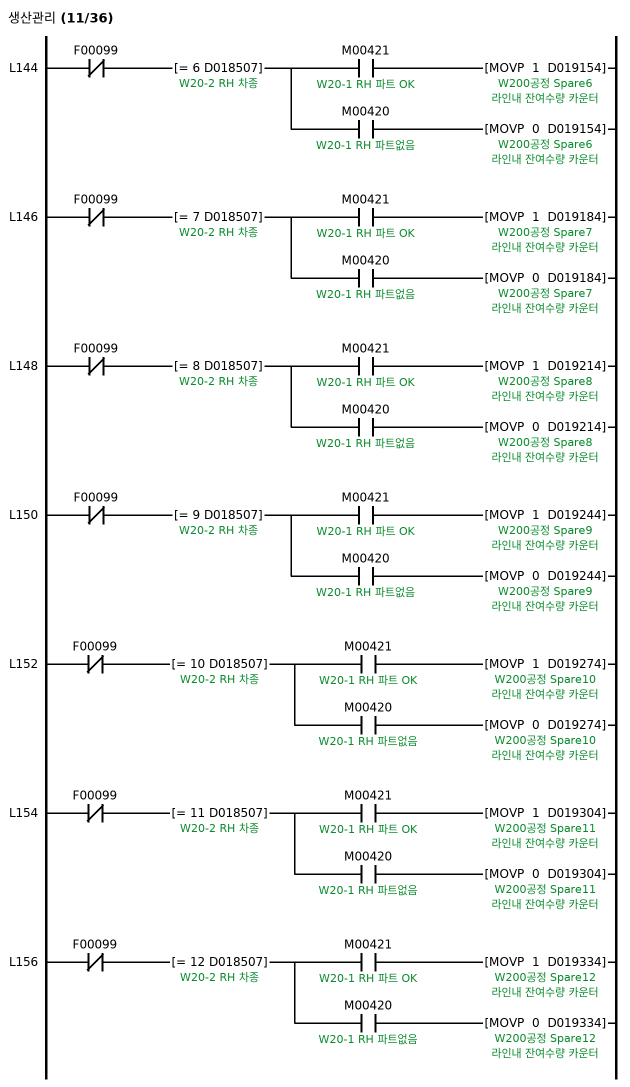
[picture p456: 생산관리 rungs L144-L156]
; L144
LOAD NOT  F00099
AND=      6 D018507	// W20-2 RH 차종
MPUSH
AND       M00421	// W20-1 RH 파트 OK
MOVP      1 D019154	// W200공정 Spare6 라인내 잔여수량 카운터
MPOP
AND       M00420	// W20-1 RH 파트없음
MOVP      0 D019154	// W200공정 Spare6 라인내 잔여수량 카운터
; L146
LOAD NOT  F00099
AND=      7 D018507	// W20-2 RH 차종
MPUSH
AND       M00421	// W20-1 RH 파트 OK
MOVP      1 D019184	// W200공정 Spare7 라인내 잔여수량 카운터
MPOP
AND       M00420	// W20-1 RH 파트없음
MOVP      0 D019184	// W200공정 Spare7 라인내 잔여수량 카운터
; L148
LOAD NOT  F00099
AND=      8 D018507	// W20-2 RH 차종
MPUSH
AND       M00421	// W20-1 RH 파트 OK
MOVP      1 D019214	// W200공정 Spare8 라인내 잔여수량 카운터
MPOP
AND       M00420	// W20-1 RH 파트없음
MOVP      0 D019214	// W200공정 Spare8 라인내 잔여수량 카운터
; L150
LOAD NOT  F00099
AND=      9 D018507	// W20-2 RH 차종
MPUSH
AND       M00421	// W20-1 RH 파트 OK
MOVP      1 D019244	// W200공정 Spare9 라인내 잔여수량 카운터
MPOP
AND       M00420	// W20-1 RH 파트없음
MOVP      0 D019244	// W200공정 Spare9 라인내 잔여수량 카운터
; L152
LOAD NOT  F00099
AND=      10 D018507	// W20-2 RH 차종
MPUSH
AND       M00421	// W20-1 RH 파트 OK
MOVP      1 D019274	// W200공정 Spare10 라인내 잔여수량 카운터
MPOP
AND       M00420	// W20-1 RH 파트없음
MOVP      0 D019274	// W200공정 Spare10 라인내 잔여수량 카운터
; L154
LOAD NOT  F00099
AND=      11 D018507	// W20-2 RH 차종
MPUSH
AND       M00421	// W20-1 RH 파트 OK
MOVP      1 D019304	// W200공정 Spare11 라인내 잔여수량 카운터
MPOP
AND       M00420	// W20-1 RH 파트없음
MOVP      0 D019304	// W200공정 Spare11 라인내 잔여수량 카운터
; L156
LOAD NOT  F00099
AND=      12 D018507	// W20-2 RH 차종
MPUSH
AND       M00421	// W20-1 RH 파트 OK
MOVP      1 D019334	// W200공정 Spare12 라인내 잔여수량 카운터
MPOP
AND       M00420	// W20-1 RH 파트없음
MOVP      0 D019334	// W200공정 Spare12 라인내 잔여수량 카운터

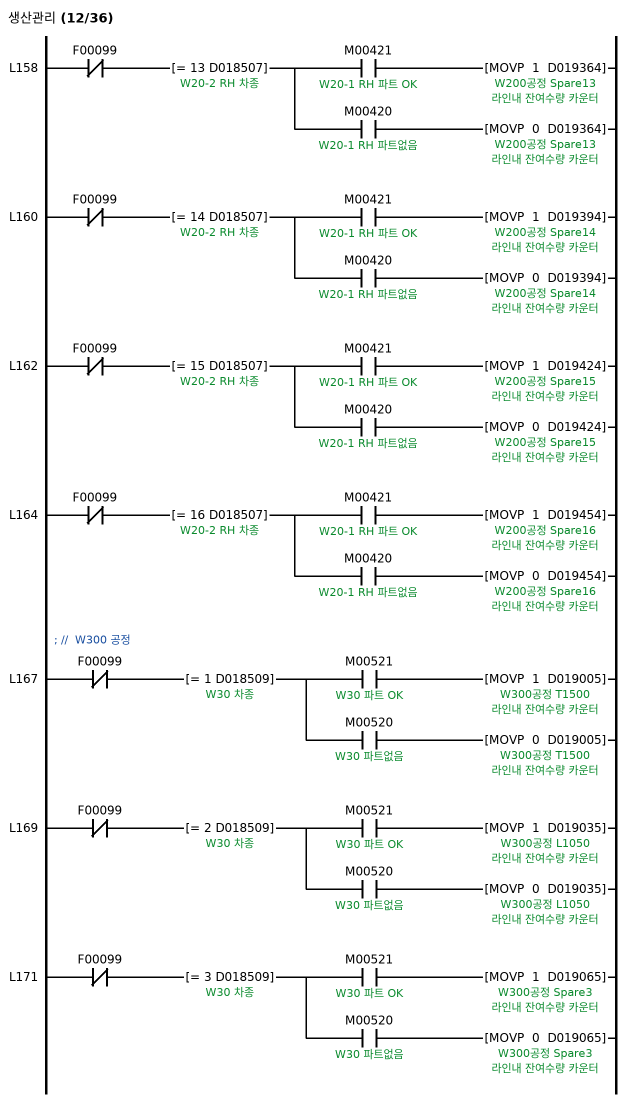
; L158
LOAD NOT  F00099
AND=      13 D018507	// W20-2 RH 차종
MPUSH
AND       M00421	// W20-1 RH 파트 OK
MOVP      1 D019364	// W200공정 Spare13 라인내 잔여수량 카운터
MPOP
AND       M00420	// W20-1 RH 파트없음
MOVP      0 D019364	// W200공정 Spare13 라인내 잔여수량 카운터
; L160
LOAD NOT  F00099
AND=      14 D018507	// W20-2 RH 차종
MPUSH
AND       M00421	// W20-1 RH 파트 OK
MOVP      1 D019394	// W200공정 Spare14 라인내 잔여수량 카운터
MPOP
AND       M00420	// W20-1 RH 파트없음
MOVP      0 D019394	// W200공정 Spare14 라인내 잔여수량 카운터
; L162
LOAD NOT  F00099
AND=      15 D018507	// W20-2 RH 차종
MPUSH
AND       M00421	// W20-1 RH 파트 OK
MOVP      1 D019424	// W200공정 Spare15 라인내 잔여수량 카운터
MPOP
AND       M00420	// W20-1 RH 파트없음
MOVP      0 D019424	// W200공정 Spare15 라인내 잔여수량 카운터
; L164
LOAD NOT  F00099
AND=      16 D018507	// W20-2 RH 차종
MPUSH
AND       M00421	// W20-1 RH 파트 OK
MOVP      1 D019454	// W200공정 Spare16 라인내 잔여수량 카운터
MPOP
AND       M00420	// W20-1 RH 파트없음
MOVP      0 D019454	// W200공정 Spare16 라인내 잔여수량 카운터
//   //  W300 공정
; L167
LOAD NOT  F00099
AND=      1 D018509	// W30 차종
MPUSH
AND       M00521	// W30 파트 OK
MOVP      1 D019005	// W300공정 T1500 라인내 잔여수량 카운터
MPOP
AND       M00520	// W30 파트없음
MOVP      0 D019005	// W300공정 T1500 라인내 잔여수량 카운터
; L169
LOAD NOT  F00099
AND=      2 D018509	// W30 차종
MPUSH
AND       M00521	// W30 파트 OK
MOVP      1 D019035	// W300공정 L1050 라인내 잔여수량 카운터
MPOP
AND       M00520	// W30 파트없음
MOVP      0 D019035	// W300공정 L1050 라인내 잔여수량 카운터
; L171
LOAD NOT  F00099
AND=      3 D018509	// W30 차종
MPUSH
AND       M00521	// W30 파트 OK
MOVP      1 D019065	// W300공정 Spare3 라인내 잔여수량 카운터
MPOP
AND       M00520	// W30 파트없음
MOVP      0 D019065	// W300공정 Spare3 라인내 잔여수량 카운터

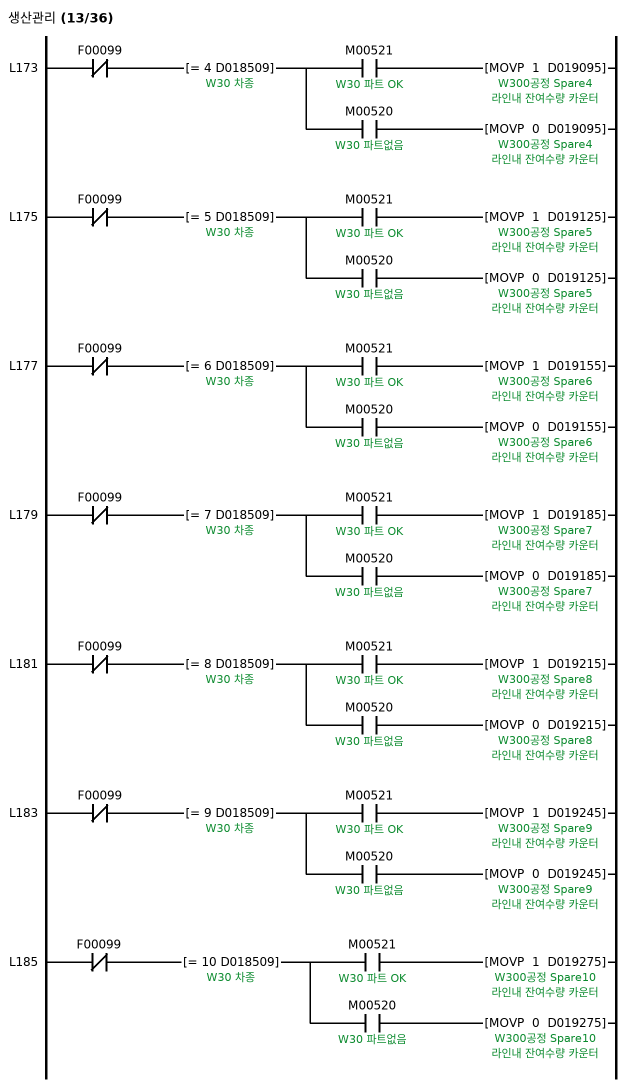
; L173
LOAD NOT  F00099
AND=      4 D018509	// W30 차종
MPUSH
AND       M00521	// W30 파트 OK
MOVP      1 D019095	// W300공정 Spare4 라인내 잔여수량 카운터
MPOP
AND       M00520	// W30 파트없음
MOVP      0 D019095	// W300공정 Spare4 라인내 잔여수량 카운터
; L175
LOAD NOT  F00099
AND=      5 D018509	// W30 차종
MPUSH
AND       M00521	// W30 파트 OK
MOVP      1 D019125	// W300공정 Spare5 라인내 잔여수량 카운터
MPOP
AND       M00520	// W30 파트없음
MOVP      0 D019125	// W300공정 Spare5 라인내 잔여수량 카운터
; L177
LOAD NOT  F00099
AND=      6 D018509	// W30 차종
MPUSH
AND       M00521	// W30 파트 OK
MOVP      1 D019155	// W300공정 Spare6 라인내 잔여수량 카운터
MPOP
AND       M00520	// W30 파트없음
MOVP      0 D019155	// W300공정 Spare6 라인내 잔여수량 카운터
; L179
LOAD NOT  F00099
AND=      7 D018509	// W30 차종
MPUSH
AND       M00521	// W30 파트 OK
MOVP      1 D019185	// W300공정 Spare7 라인내 잔여수량 카운터
MPOP
AND       M00520	// W30 파트없음
MOVP      0 D019185	// W300공정 Spare7 라인내 잔여수량 카운터
; L181
LOAD NOT  F00099
AND=      8 D018509	// W30 차종
MPUSH
AND       M00521	// W30 파트 OK
MOVP      1 D019215	// W300공정 Spare8 라인내 잔여수량 카운터
MPOP
AND       M00520	// W30 파트없음
MOVP      0 D019215	// W300공정 Spare8 라인내 잔여수량 카운터
; L183
LOAD NOT  F00099
AND=      9 D018509	// W30 차종
MPUSH
AND       M00521	// W30 파트 OK
MOVP      1 D019245	// W300공정 Spare9 라인내 잔여수량 카운터
MPOP
AND       M00520	// W30 파트없음
MOVP      0 D019245	// W300공정 Spare9 라인내 잔여수량 카운터
; L185
LOAD NOT  F00099
AND=      10 D018509	// W30 차종
MPUSH
AND       M00521	// W30 파트 OK
MOVP      1 D019275	// W300공정 Spare10 라인내 잔여수량 카운터
MPOP
AND       M00520	// W30 파트없음
MOVP      0 D019275	// W300공정 Spare10 라인내 잔여수량 카운터

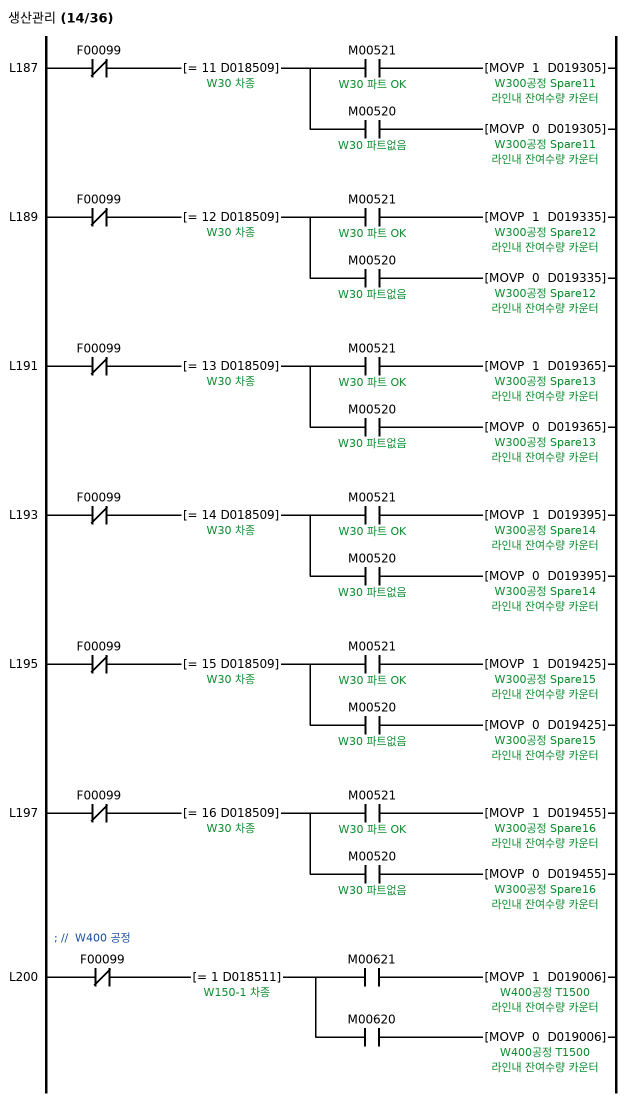
; L187
LOAD NOT  F00099
AND=      11 D018509	// W30 차종
MPUSH
AND       M00521	// W30 파트 OK
MOVP      1 D019305	// W300공정 Spare11 라인내 잔여수량 카운터
MPOP
AND       M00520	// W30 파트없음
MOVP      0 D019305	// W300공정 Spare11 라인내 잔여수량 카운터
; L189
LOAD NOT  F00099
AND=      12 D018509	// W30 차종
MPUSH
AND       M00521	// W30 파트 OK
MOVP      1 D019335	// W300공정 Spare12 라인내 잔여수량 카운터
MPOP
AND       M00520	// W30 파트없음
MOVP      0 D019335	// W300공정 Spare12 라인내 잔여수량 카운터
; L191
LOAD NOT  F00099
AND=      13 D018509	// W30 차종
MPUSH
AND       M00521	// W30 파트 OK
MOVP      1 D019365	// W300공정 Spare13 라인내 잔여수량 카운터
MPOP
AND       M00520	// W30 파트없음
MOVP      0 D019365	// W300공정 Spare13 라인내 잔여수량 카운터
; L193
LOAD NOT  F00099
AND=      14 D018509	// W30 차종
MPUSH
AND       M00521	// W30 파트 OK
MOVP      1 D019395	// W300공정 Spare14 라인내 잔여수량 카운터
MPOP
AND       M00520	// W30 파트없음
MOVP      0 D019395	// W300공정 Spare14 라인내 잔여수량 카운터
; L195
LOAD NOT  F00099
AND=      15 D018509	// W30 차종
MPUSH
AND       M00521	// W30 파트 OK
MOVP      1 D019425	// W300공정 Spare15 라인내 잔여수량 카운터
MPOP
AND       M00520	// W30 파트없음
MOVP      0 D019425	// W300공정 Spare15 라인내 잔여수량 카운터
; L197
LOAD NOT  F00099
AND=      16 D018509	// W30 차종
MPUSH
AND       M00521	// W30 파트 OK
MOVP      1 D019455	// W300공정 Spare16 라인내 잔여수량 카운터
MPOP
AND       M00520	// W30 파트없음
MOVP      0 D019455	// W300공정 Spare16 라인내 잔여수량 카운터
//   //  W400 공정
; L200
LOAD NOT  F00099
AND=      1 D018511	// W150-1 차종
MPUSH
AND       M00621
MOVP      1 D019006	// W400공정 T1500 라인내 잔여수량 카운터
MPOP
AND       M00620
MOVP      0 D019006	// W400공정 T1500 라인내 잔여수량 카운터

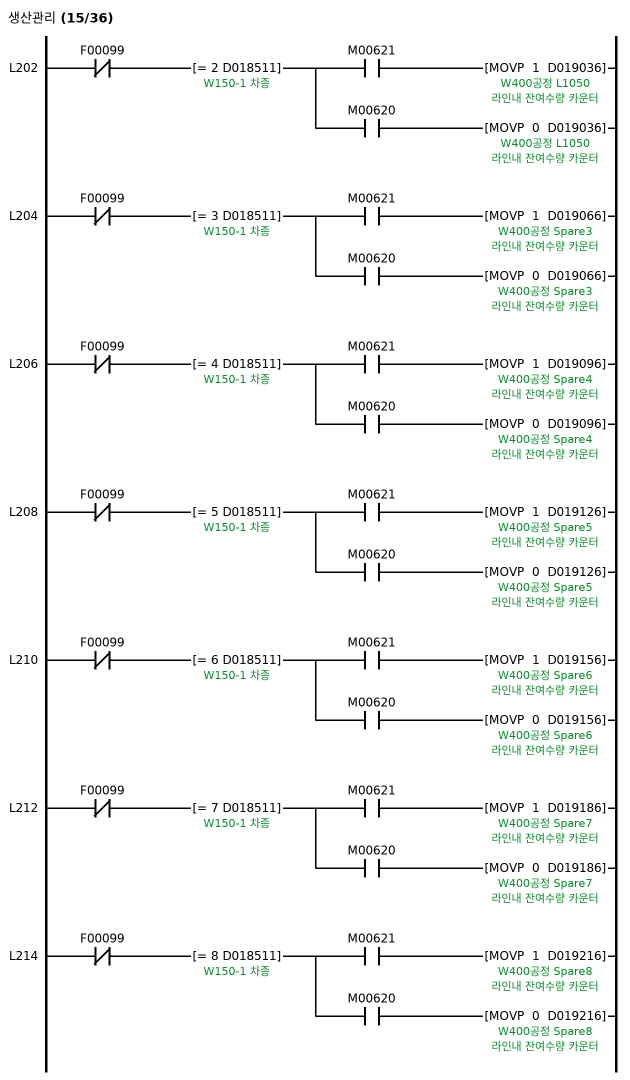
; L202
LOAD NOT  F00099
AND=      2 D018511	// W150-1 차종
MPUSH
AND       M00621
MOVP      1 D019036	// W400공정 L1050 라인내 잔여수량 카운터
MPOP
AND       M00620
MOVP      0 D019036	// W400공정 L1050 라인내 잔여수량 카운터
; L204
LOAD NOT  F00099
AND=      3 D018511	// W150-1 차종
MPUSH
AND       M00621
MOVP      1 D019066	// W400공정 Spare3 라인내 잔여수량 카운터
MPOP
AND       M00620
MOVP      0 D019066	// W400공정 Spare3 라인내 잔여수량 카운터
; L206
LOAD NOT  F00099
AND=      4 D018511	// W150-1 차종
MPUSH
AND       M00621
MOVP      1 D019096	// W400공정 Spare4 라인내 잔여수량 카운터
MPOP
AND       M00620
MOVP      0 D019096	// W400공정 Spare4 라인내 잔여수량 카운터
; L208
LOAD NOT  F00099
AND=      5 D018511	// W150-1 차종
MPUSH
AND       M00621
MOVP      1 D019126	// W400공정 Spare5 라인내 잔여수량 카운터
MPOP
AND       M00620
MOVP      0 D019126	// W400공정 Spare5 라인내 잔여수량 카운터
; L210
LOAD NOT  F00099
AND=      6 D018511	// W150-1 차종
MPUSH
AND       M00621
MOVP      1 D019156	// W400공정 Spare6 라인내 잔여수량 카운터
MPOP
AND       M00620
MOVP      0 D019156	// W400공정 Spare6 라인내 잔여수량 카운터
; L212
LOAD NOT  F00099
AND=      7 D018511	// W150-1 차종
MPUSH
AND       M00621
MOVP      1 D019186	// W400공정 Spare7 라인내 잔여수량 카운터
MPOP
AND       M00620
MOVP      0 D019186	// W400공정 Spare7 라인내 잔여수량 카운터
; L214
LOAD NOT  F00099
AND=      8 D018511	// W150-1 차종
MPUSH
AND       M00621
MOVP      1 D019216	// W400공정 Spare8 라인내 잔여수량 카운터
MPOP
AND       M00620
MOVP      0 D019216	// W400공정 Spare8 라인내 잔여수량 카운터

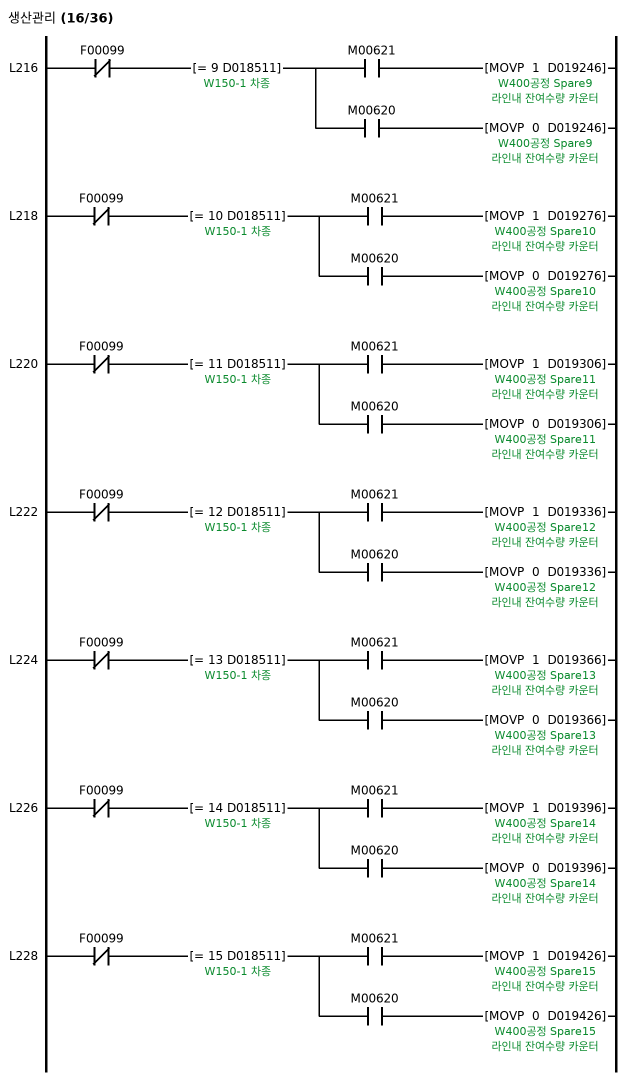
; L216
LOAD NOT  F00099
AND=      9 D018511	// W150-1 차종
MPUSH
AND       M00621
MOVP      1 D019246	// W400공정 Spare9 라인내 잔여수량 카운터
MPOP
AND       M00620
MOVP      0 D019246	// W400공정 Spare9 라인내 잔여수량 카운터
; L218
LOAD NOT  F00099
AND=      10 D018511	// W150-1 차종
MPUSH
AND       M00621
MOVP      1 D019276	// W400공정 Spare10 라인내 잔여수량 카운터
MPOP
AND       M00620
MOVP      0 D019276	// W400공정 Spare10 라인내 잔여수량 카운터
; L220
LOAD NOT  F00099
AND=      11 D018511	// W150-1 차종
MPUSH
AND       M00621
MOVP      1 D019306	// W400공정 Spare11 라인내 잔여수량 카운터
MPOP
AND       M00620
MOVP      0 D019306	// W400공정 Spare11 라인내 잔여수량 카운터
; L222
LOAD NOT  F00099
AND=      12 D018511	// W150-1 차종
MPUSH
AND       M00621
MOVP      1 D019336	// W400공정 Spare12 라인내 잔여수량 카운터
MPOP
AND       M00620
MOVP      0 D019336	// W400공정 Spare12 라인내 잔여수량 카운터
; L224
LOAD NOT  F00099
AND=      13 D018511	// W150-1 차종
MPUSH
AND       M00621
MOVP      1 D019366	// W400공정 Spare13 라인내 잔여수량 카운터
MPOP
AND       M00620
MOVP      0 D019366	// W400공정 Spare13 라인내 잔여수량 카운터
; L226
LOAD NOT  F00099
AND=      14 D018511	// W150-1 차종
MPUSH
AND       M00621
MOVP      1 D019396	// W400공정 Spare14 라인내 잔여수량 카운터
MPOP
AND       M00620
MOVP      0 D019396	// W400공정 Spare14 라인내 잔여수량 카운터
; L228
LOAD NOT  F00099
AND=      15 D018511	// W150-1 차종
MPUSH
AND       M00621
MOVP      1 D019426	// W400공정 Spare15 라인내 잔여수량 카운터
MPOP
AND       M00620
MOVP      0 D019426	// W400공정 Spare15 라인내 잔여수량 카운터

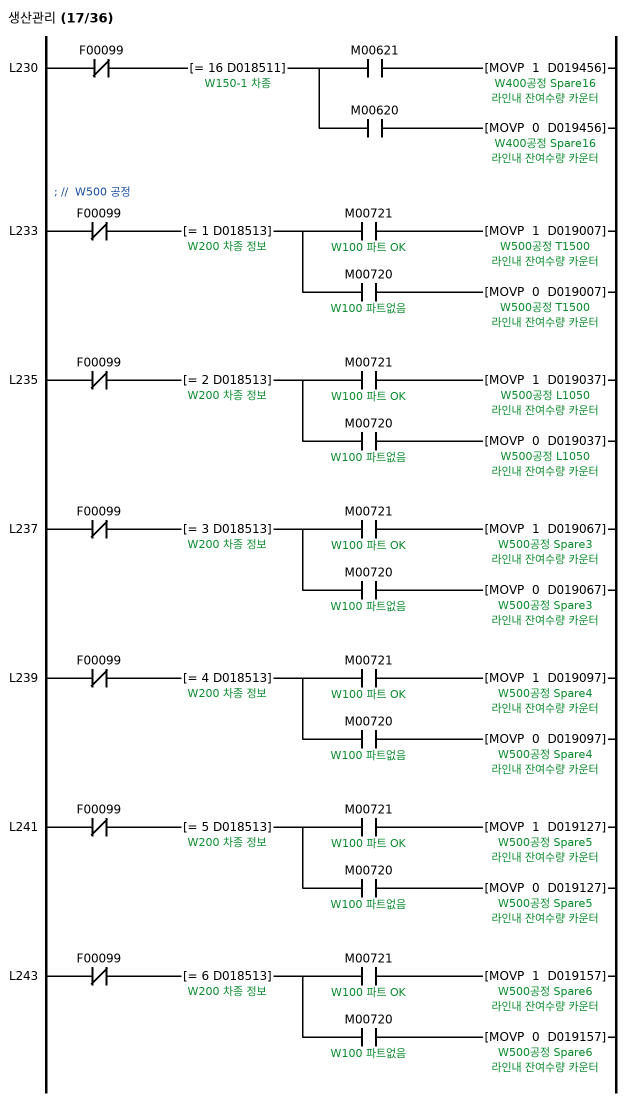
; L230
LOAD NOT  F00099
AND=      16 D018511	// W150-1 차종
MPUSH
AND       M00621
MOVP      1 D019456	// W400공정 Spare16 라인내 잔여수량 카운터
MPOP
AND       M00620
MOVP      0 D019456	// W400공정 Spare16 라인내 잔여수량 카운터
//   //  W500 공정
; L233
LOAD NOT  F00099
AND=      1 D018513	// W200 차종 정보
MPUSH
AND       M00721	// W100 파트 OK
MOVP      1 D019007	// W500공정 T1500 라인내 잔여수량 카운터
MPOP
AND       M00720	// W100 파트없음
MOVP      0 D019007	// W500공정 T1500 라인내 잔여수량 카운터
; L235
LOAD NOT  F00099
AND=      2 D018513	// W200 차종 정보
MPUSH
AND       M00721	// W100 파트 OK
MOVP      1 D019037	// W500공정 L1050 라인내 잔여수량 카운터
MPOP
AND       M00720	// W100 파트없음
MOVP      0 D019037	// W500공정 L1050 라인내 잔여수량 카운터
; L237
LOAD NOT  F00099
AND=      3 D018513	// W200 차종 정보
MPUSH
AND       M00721	// W100 파트 OK
MOVP      1 D019067	// W500공정 Spare3 라인내 잔여수량 카운터
MPOP
AND       M00720	// W100 파트없음
MOVP      0 D019067	// W500공정 Spare3 라인내 잔여수량 카운터
; L239
LOAD NOT  F00099
AND=      4 D018513	// W200 차종 정보
MPUSH
AND       M00721	// W100 파트 OK
MOVP      1 D019097	// W500공정 Spare4 라인내 잔여수량 카운터
MPOP
AND       M00720	// W100 파트없음
MOVP      0 D019097	// W500공정 Spare4 라인내 잔여수량 카운터
; L241
LOAD NOT  F00099
AND=      5 D018513	// W200 차종 정보
MPUSH
AND       M00721	// W100 파트 OK
MOVP      1 D019127	// W500공정 Spare5 라인내 잔여수량 카운터
MPOP
AND       M00720	// W100 파트없음
MOVP      0 D019127	// W500공정 Spare5 라인내 잔여수량 카운터
; L243
LOAD NOT  F00099
AND=      6 D018513	// W200 차종 정보
MPUSH
AND       M00721	// W100 파트 OK
MOVP      1 D019157	// W500공정 Spare6 라인내 잔여수량 카운터
MPOP
AND       M00720	// W100 파트없음
MOVP      0 D019157	// W500공정 Spare6 라인내 잔여수량 카운터

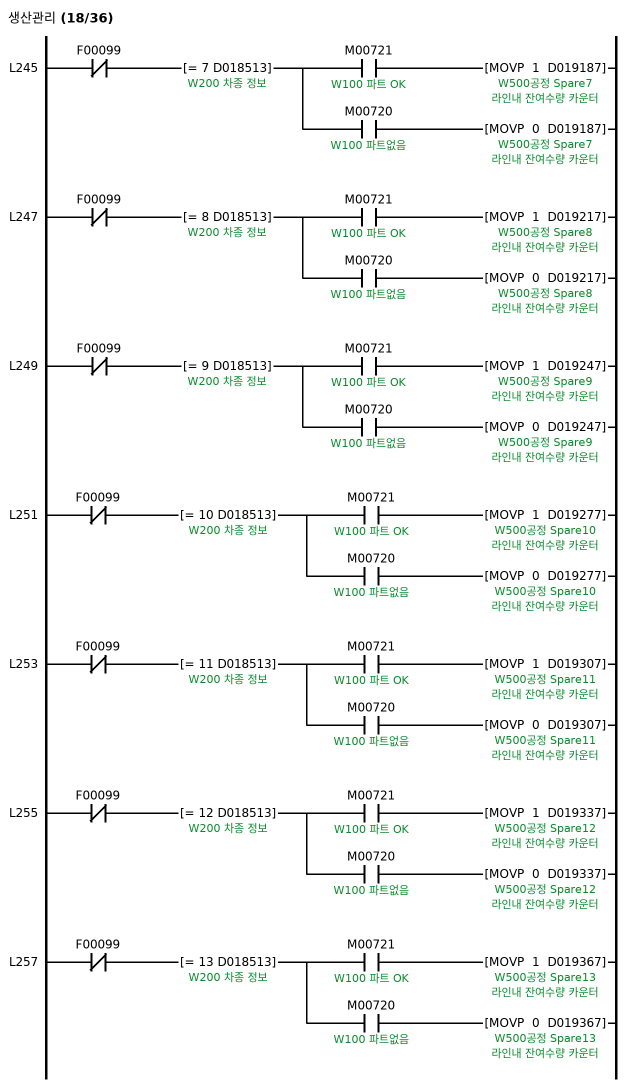
; L245
LOAD NOT  F00099
AND=      7 D018513	// W200 차종 정보
MPUSH
AND       M00721	// W100 파트 OK
MOVP      1 D019187	// W500공정 Spare7 라인내 잔여수량 카운터
MPOP
AND       M00720	// W100 파트없음
MOVP      0 D019187	// W500공정 Spare7 라인내 잔여수량 카운터
; L247
LOAD NOT  F00099
AND=      8 D018513	// W200 차종 정보
MPUSH
AND       M00721	// W100 파트 OK
MOVP      1 D019217	// W500공정 Spare8 라인내 잔여수량 카운터
MPOP
AND       M00720	// W100 파트없음
MOVP      0 D019217	// W500공정 Spare8 라인내 잔여수량 카운터
; L249
LOAD NOT  F00099
AND=      9 D018513	// W200 차종 정보
MPUSH
AND       M00721	// W100 파트 OK
MOVP      1 D019247	// W500공정 Spare9 라인내 잔여수량 카운터
MPOP
AND       M00720	// W100 파트없음
MOVP      0 D019247	// W500공정 Spare9 라인내 잔여수량 카운터
; L251
LOAD NOT  F00099
AND=      10 D018513	// W200 차종 정보
MPUSH
AND       M00721	// W100 파트 OK
MOVP      1 D019277	// W500공정 Spare10 라인내 잔여수량 카운터
MPOP
AND       M00720	// W100 파트없음
MOVP      0 D019277	// W500공정 Spare10 라인내 잔여수량 카운터
; L253
LOAD NOT  F00099
AND=      11 D018513	// W200 차종 정보
MPUSH
AND       M00721	// W100 파트 OK
MOVP      1 D019307	// W500공정 Spare11 라인내 잔여수량 카운터
MPOP
AND       M00720	// W100 파트없음
MOVP      0 D019307	// W500공정 Spare11 라인내 잔여수량 카운터
; L255
LOAD NOT  F00099
AND=      12 D018513	// W200 차종 정보
MPUSH
AND       M00721	// W100 파트 OK
MOVP      1 D019337	// W500공정 Spare12 라인내 잔여수량 카운터
MPOP
AND       M00720	// W100 파트없음
MOVP      0 D019337	// W500공정 Spare12 라인내 잔여수량 카운터
; L257
LOAD NOT  F00099
AND=      13 D018513	// W200 차종 정보
MPUSH
AND       M00721	// W100 파트 OK
MOVP      1 D019367	// W500공정 Spare13 라인내 잔여수량 카운터
MPOP
AND       M00720	// W100 파트없음
MOVP      0 D019367	// W500공정 Spare13 라인내 잔여수량 카운터

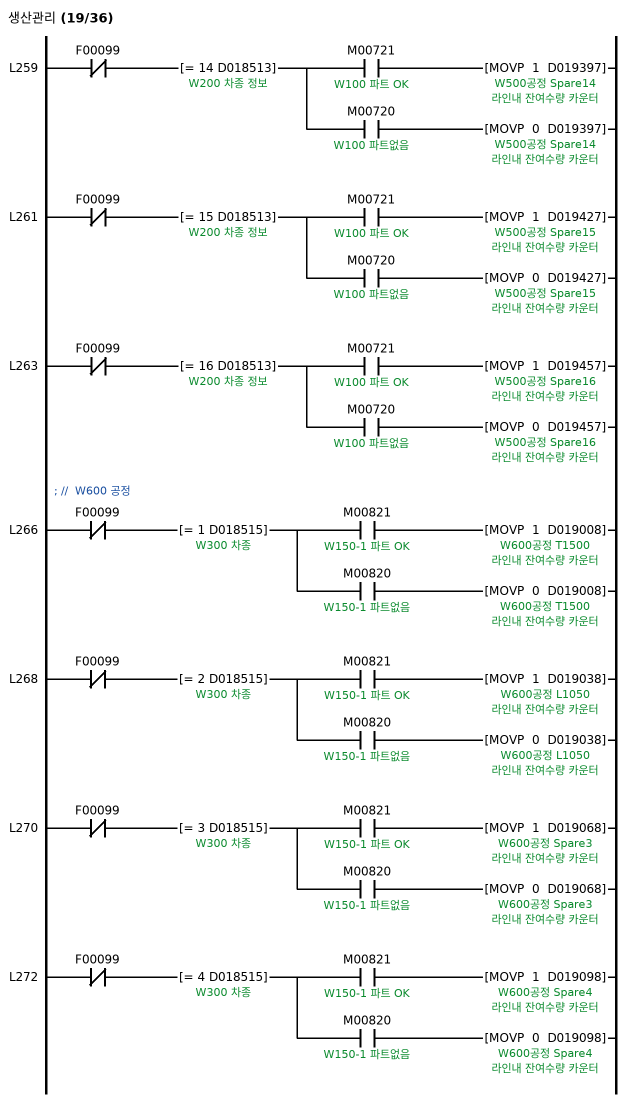
; L259
LOAD NOT  F00099
AND=      14 D018513	// W200 차종 정보
MPUSH
AND       M00721	// W100 파트 OK
MOVP      1 D019397	// W500공정 Spare14 라인내 잔여수량 카운터
MPOP
AND       M00720	// W100 파트없음
MOVP      0 D019397	// W500공정 Spare14 라인내 잔여수량 카운터
; L261
LOAD NOT  F00099
AND=      15 D018513	// W200 차종 정보
MPUSH
AND       M00721	// W100 파트 OK
MOVP      1 D019427	// W500공정 Spare15 라인내 잔여수량 카운터
MPOP
AND       M00720	// W100 파트없음
MOVP      0 D019427	// W500공정 Spare15 라인내 잔여수량 카운터
; L263
LOAD NOT  F00099
AND=      16 D018513	// W200 차종 정보
MPUSH
AND       M00721	// W100 파트 OK
MOVP      1 D019457	// W500공정 Spare16 라인내 잔여수량 카운터
MPOP
AND       M00720	// W100 파트없음
MOVP      0 D019457	// W500공정 Spare16 라인내 잔여수량 카운터
//   //  W600 공정
; L266
LOAD NOT  F00099
AND=      1 D018515	// W300 차종
MPUSH
AND       M00821	// W150-1 파트 OK
MOVP      1 D019008	// W600공정 T1500 라인내 잔여수량 카운터
MPOP
AND       M00820	// W150-1 파트없음
MOVP      0 D019008	// W600공정 T1500 라인내 잔여수량 카운터
; L268
LOAD NOT  F00099
AND=      2 D018515	// W300 차종
MPUSH
AND       M00821	// W150-1 파트 OK
MOVP      1 D019038	// W600공정 L1050 라인내 잔여수량 카운터
MPOP
AND       M00820	// W150-1 파트없음
MOVP      0 D019038	// W600공정 L1050 라인내 잔여수량 카운터
; L270
LOAD NOT  F00099
AND=      3 D018515	// W300 차종
MPUSH
AND       M00821	// W150-1 파트 OK
MOVP      1 D019068	// W600공정 Spare3 라인내 잔여수량 카운터
MPOP
AND       M00820	// W150-1 파트없음
MOVP      0 D019068	// W600공정 Spare3 라인내 잔여수량 카운터
; L272
LOAD NOT  F00099
AND=      4 D018515	// W300 차종
MPUSH
AND       M00821	// W150-1 파트 OK
MOVP      1 D019098	// W600공정 Spare4 라인내 잔여수량 카운터
MPOP
AND       M00820	// W150-1 파트없음
MOVP      0 D019098	// W600공정 Spare4 라인내 잔여수량 카운터

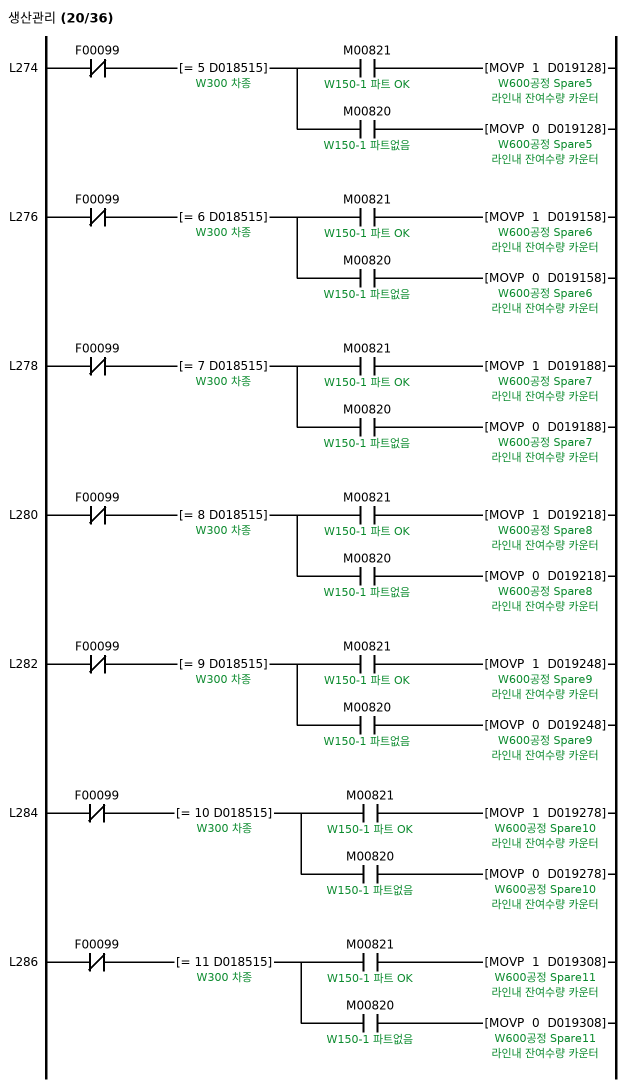
; L274
LOAD NOT  F00099
AND=      5 D018515	// W300 차종
MPUSH
AND       M00821	// W150-1 파트 OK
MOVP      1 D019128	// W600공정 Spare5 라인내 잔여수량 카운터
MPOP
AND       M00820	// W150-1 파트없음
MOVP      0 D019128	// W600공정 Spare5 라인내 잔여수량 카운터
; L276
LOAD NOT  F00099
AND=      6 D018515	// W300 차종
MPUSH
AND       M00821	// W150-1 파트 OK
MOVP      1 D019158	// W600공정 Spare6 라인내 잔여수량 카운터
MPOP
AND       M00820	// W150-1 파트없음
MOVP      0 D019158	// W600공정 Spare6 라인내 잔여수량 카운터
; L278
LOAD NOT  F00099
AND=      7 D018515	// W300 차종
MPUSH
AND       M00821	// W150-1 파트 OK
MOVP      1 D019188	// W600공정 Spare7 라인내 잔여수량 카운터
MPOP
AND       M00820	// W150-1 파트없음
MOVP      0 D019188	// W600공정 Spare7 라인내 잔여수량 카운터
; L280
LOAD NOT  F00099
AND=      8 D018515	// W300 차종
MPUSH
AND       M00821	// W150-1 파트 OK
MOVP      1 D019218	// W600공정 Spare8 라인내 잔여수량 카운터
MPOP
AND       M00820	// W150-1 파트없음
MOVP      0 D019218	// W600공정 Spare8 라인내 잔여수량 카운터
; L282
LOAD NOT  F00099
AND=      9 D018515	// W300 차종
MPUSH
AND       M00821	// W150-1 파트 OK
MOVP      1 D019248	// W600공정 Spare9 라인내 잔여수량 카운터
MPOP
AND       M00820	// W150-1 파트없음
MOVP      0 D019248	// W600공정 Spare9 라인내 잔여수량 카운터
; L284
LOAD NOT  F00099
AND=      10 D018515	// W300 차종
MPUSH
AND       M00821	// W150-1 파트 OK
MOVP      1 D019278	// W600공정 Spare10 라인내 잔여수량 카운터
MPOP
AND       M00820	// W150-1 파트없음
MOVP      0 D019278	// W600공정 Spare10 라인내 잔여수량 카운터
; L286
LOAD NOT  F00099
AND=      11 D018515	// W300 차종
MPUSH
AND       M00821	// W150-1 파트 OK
MOVP      1 D019308	// W600공정 Spare11 라인내 잔여수량 카운터
MPOP
AND       M00820	// W150-1 파트없음
MOVP      0 D019308	// W600공정 Spare11 라인내 잔여수량 카운터

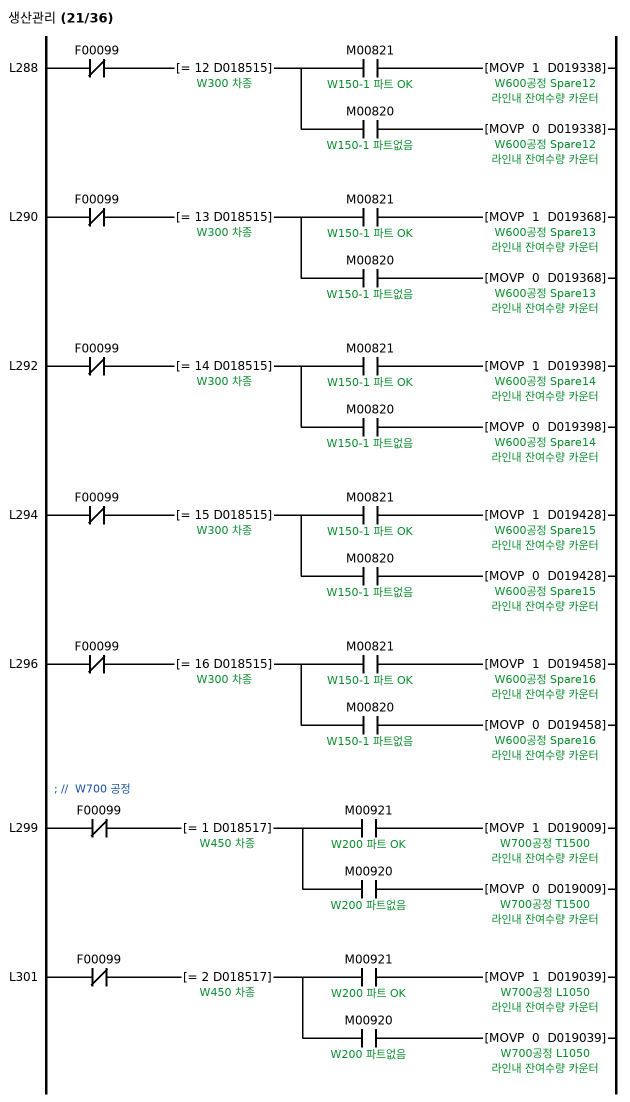
; L288
LOAD NOT  F00099
AND=      12 D018515	// W300 차종
MPUSH
AND       M00821	// W150-1 파트 OK
MOVP      1 D019338	// W600공정 Spare12 라인내 잔여수량 카운터
MPOP
AND       M00820	// W150-1 파트없음
MOVP      0 D019338	// W600공정 Spare12 라인내 잔여수량 카운터
; L290
LOAD NOT  F00099
AND=      13 D018515	// W300 차종
MPUSH
AND       M00821	// W150-1 파트 OK
MOVP      1 D019368	// W600공정 Spare13 라인내 잔여수량 카운터
MPOP
AND       M00820	// W150-1 파트없음
MOVP      0 D019368	// W600공정 Spare13 라인내 잔여수량 카운터
; L292
LOAD NOT  F00099
AND=      14 D018515	// W300 차종
MPUSH
AND       M00821	// W150-1 파트 OK
MOVP      1 D019398	// W600공정 Spare14 라인내 잔여수량 카운터
MPOP
AND       M00820	// W150-1 파트없음
MOVP      0 D019398	// W600공정 Spare14 라인내 잔여수량 카운터
; L294
LOAD NOT  F00099
AND=      15 D018515	// W300 차종
MPUSH
AND       M00821	// W150-1 파트 OK
MOVP      1 D019428	// W600공정 Spare15 라인내 잔여수량 카운터
MPOP
AND       M00820	// W150-1 파트없음
MOVP      0 D019428	// W600공정 Spare15 라인내 잔여수량 카운터
; L296
LOAD NOT  F00099
AND=      16 D018515	// W300 차종
MPUSH
AND       M00821	// W150-1 파트 OK
MOVP      1 D019458	// W600공정 Spare16 라인내 잔여수량 카운터
MPOP
AND       M00820	// W150-1 파트없음
MOVP      0 D019458	// W600공정 Spare16 라인내 잔여수량 카운터
//   //  W700 공정
; L299
LOAD NOT  F00099
AND=      1 D018517	// W450 차종
MPUSH
AND       M00921	// W200 파트 OK
MOVP      1 D019009	// W700공정 T1500 라인내 잔여수량 카운터
MPOP
AND       M00920	// W200 파트없음
MOVP      0 D019009	// W700공정 T1500 라인내 잔여수량 카운터
; L301
LOAD NOT  F00099
AND=      2 D018517	// W450 차종
MPUSH
AND       M00921	// W200 파트 OK
MOVP      1 D019039	// W700공정 L1050 라인내 잔여수량 카운터
MPOP
AND       M00920	// W200 파트없음
MOVP      0 D019039	// W700공정 L1050 라인내 잔여수량 카운터

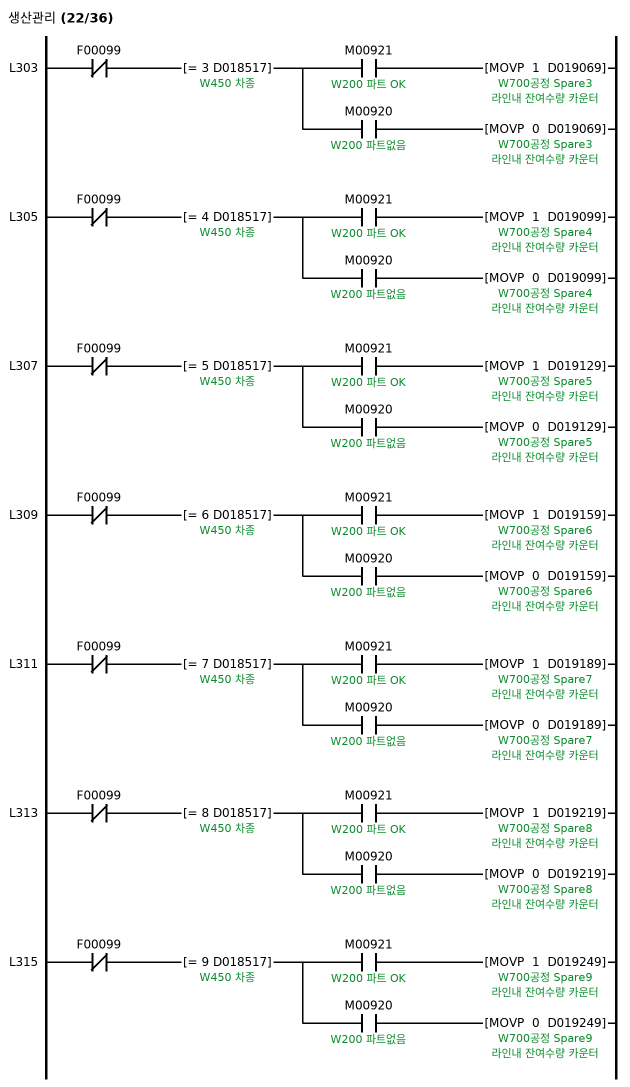
; L303
LOAD NOT  F00099
AND=      3 D018517	// W450 차종
MPUSH
AND       M00921	// W200 파트 OK
MOVP      1 D019069	// W700공정 Spare3 라인내 잔여수량 카운터
MPOP
AND       M00920	// W200 파트없음
MOVP      0 D019069	// W700공정 Spare3 라인내 잔여수량 카운터
; L305
LOAD NOT  F00099
AND=      4 D018517	// W450 차종
MPUSH
AND       M00921	// W200 파트 OK
MOVP      1 D019099	// W700공정 Spare4 라인내 잔여수량 카운터
MPOP
AND       M00920	// W200 파트없음
MOVP      0 D019099	// W700공정 Spare4 라인내 잔여수량 카운터
; L307
LOAD NOT  F00099
AND=      5 D018517	// W450 차종
MPUSH
AND       M00921	// W200 파트 OK
MOVP      1 D019129	// W700공정 Spare5 라인내 잔여수량 카운터
MPOP
AND       M00920	// W200 파트없음
MOVP      0 D019129	// W700공정 Spare5 라인내 잔여수량 카운터
; L309
LOAD NOT  F00099
AND=      6 D018517	// W450 차종
MPUSH
AND       M00921	// W200 파트 OK
MOVP      1 D019159	// W700공정 Spare6 라인내 잔여수량 카운터
MPOP
AND       M00920	// W200 파트없음
MOVP      0 D019159	// W700공정 Spare6 라인내 잔여수량 카운터
; L311
LOAD NOT  F00099
AND=      7 D018517	// W450 차종
MPUSH
AND       M00921	// W200 파트 OK
MOVP      1 D019189	// W700공정 Spare7 라인내 잔여수량 카운터
MPOP
AND       M00920	// W200 파트없음
MOVP      0 D019189	// W700공정 Spare7 라인내 잔여수량 카운터
; L313
LOAD NOT  F00099
AND=      8 D018517	// W450 차종
MPUSH
AND       M00921	// W200 파트 OK
MOVP      1 D019219	// W700공정 Spare8 라인내 잔여수량 카운터
MPOP
AND       M00920	// W200 파트없음
MOVP      0 D019219	// W700공정 Spare8 라인내 잔여수량 카운터
; L315
LOAD NOT  F00099
AND=      9 D018517	// W450 차종
MPUSH
AND       M00921	// W200 파트 OK
MOVP      1 D019249	// W700공정 Spare9 라인내 잔여수량 카운터
MPOP
AND       M00920	// W200 파트없음
MOVP      0 D019249	// W700공정 Spare9 라인내 잔여수량 카운터

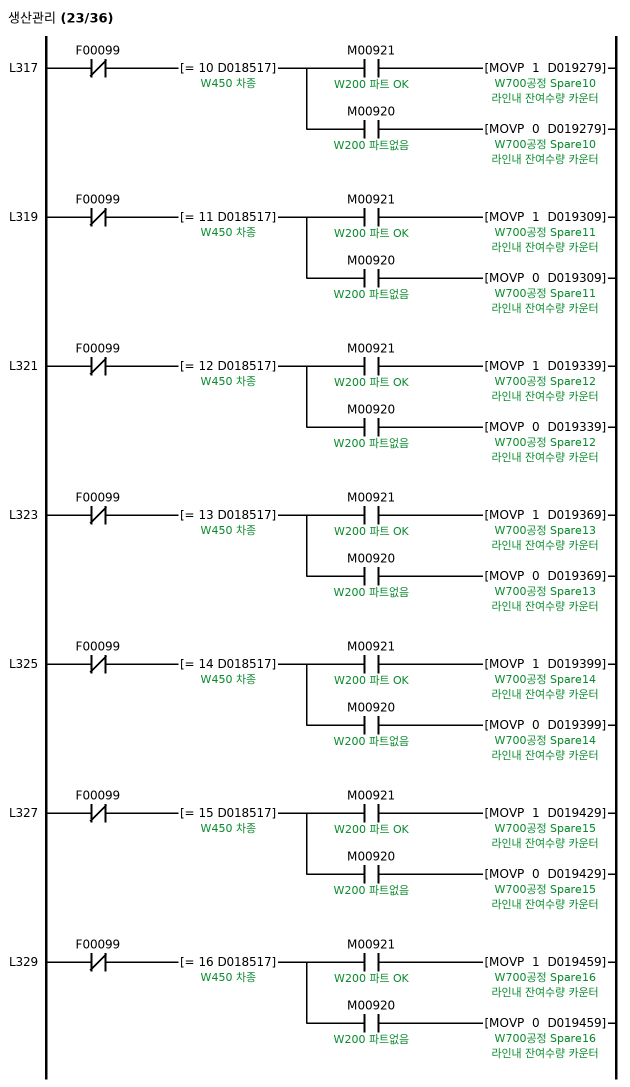
; L317
LOAD NOT  F00099
AND=      10 D018517	// W450 차종
MPUSH
AND       M00921	// W200 파트 OK
MOVP      1 D019279	// W700공정 Spare10 라인내 잔여수량 카운터
MPOP
AND       M00920	// W200 파트없음
MOVP      0 D019279	// W700공정 Spare10 라인내 잔여수량 카운터
; L319
LOAD NOT  F00099
AND=      11 D018517	// W450 차종
MPUSH
AND       M00921	// W200 파트 OK
MOVP      1 D019309	// W700공정 Spare11 라인내 잔여수량 카운터
MPOP
AND       M00920	// W200 파트없음
MOVP      0 D019309	// W700공정 Spare11 라인내 잔여수량 카운터
; L321
LOAD NOT  F00099
AND=      12 D018517	// W450 차종
MPUSH
AND       M00921	// W200 파트 OK
MOVP      1 D019339	// W700공정 Spare12 라인내 잔여수량 카운터
MPOP
AND       M00920	// W200 파트없음
MOVP      0 D019339	// W700공정 Spare12 라인내 잔여수량 카운터
; L323
LOAD NOT  F00099
AND=      13 D018517	// W450 차종
MPUSH
AND       M00921	// W200 파트 OK
MOVP      1 D019369	// W700공정 Spare13 라인내 잔여수량 카운터
MPOP
AND       M00920	// W200 파트없음
MOVP      0 D019369	// W700공정 Spare13 라인내 잔여수량 카운터
; L325
LOAD NOT  F00099
AND=      14 D018517	// W450 차종
MPUSH
AND       M00921	// W200 파트 OK
MOVP      1 D019399	// W700공정 Spare14 라인내 잔여수량 카운터
MPOP
AND       M00920	// W200 파트없음
MOVP      0 D019399	// W700공정 Spare14 라인내 잔여수량 카운터
; L327
LOAD NOT  F00099
AND=      15 D018517	// W450 차종
MPUSH
AND       M00921	// W200 파트 OK
MOVP      1 D019429	// W700공정 Spare15 라인내 잔여수량 카운터
MPOP
AND       M00920	// W200 파트없음
MOVP      0 D019429	// W700공정 Spare15 라인내 잔여수량 카운터
; L329
LOAD NOT  F00099
AND=      16 D018517	// W450 차종
MPUSH
AND       M00921	// W200 파트 OK
MOVP      1 D019459	// W700공정 Spare16 라인내 잔여수량 카운터
MPOP
AND       M00920	// W200 파트없음
MOVP      0 D019459	// W700공정 Spare16 라인내 잔여수량 카운터

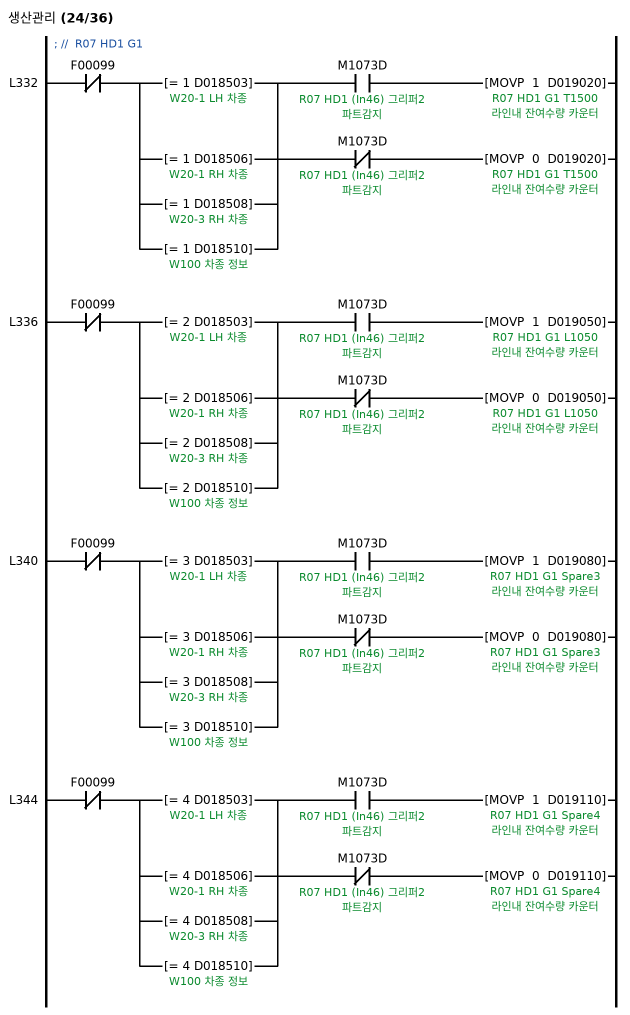
//   //  R07 HD1 G1
; L332
LOAD NOT  F00099
LOAD=     1 D018503	// W20-1 LH 차종
OR=       1 D018506	// W20-1 RH 차종
OR=       1 D018508	// W20-3 RH 차종
OR=       1 D018510	// W100 차종 정보
AND LOAD
MPUSH
AND       M1073D	// R07 HD1 (In46) 그리퍼2 파트감지
MOVP      1 D019020	// R07 HD1 G1 T1500 라인내 잔여수량 카운터
MPOP
AND NOT   M1073D	// R07 HD1 (In46) 그리퍼2 파트감지
MOVP      0 D019020	// R07 HD1 G1 T1500 라인내 잔여수량 카운터
; L336
LOAD NOT  F00099
LOAD=     2 D018503	// W20-1 LH 차종
OR=       2 D018506	// W20-1 RH 차종
OR=       2 D018508	// W20-3 RH 차종
OR=       2 D018510	// W100 차종 정보
AND LOAD
MPUSH
AND       M1073D	// R07 HD1 (In46) 그리퍼2 파트감지
MOVP      1 D019050	// R07 HD1 G1 L1050 라인내 잔여수량 카운터
MPOP
AND NOT   M1073D	// R07 HD1 (In46) 그리퍼2 파트감지
MOVP      0 D019050	// R07 HD1 G1 L1050 라인내 잔여수량 카운터
; L340
LOAD NOT  F00099
LOAD=     3 D018503	// W20-1 LH 차종
OR=       3 D018506	// W20-1 RH 차종
OR=       3 D018508	// W20-3 RH 차종
OR=       3 D018510	// W100 차종 정보
AND LOAD
MPUSH
AND       M1073D	// R07 HD1 (In46) 그리퍼2 파트감지
MOVP      1 D019080	// R07 HD1 G1 Spare3 라인내 잔여수량 카운터
MPOP
AND NOT   M1073D	// R07 HD1 (In46) 그리퍼2 파트감지
MOVP      0 D019080	// R07 HD1 G1 Spare3 라인내 잔여수량 카운터
; L344
LOAD NOT  F00099
LOAD=     4 D018503	// W20-1 LH 차종
OR=       4 D018506	// W20-1 RH 차종
OR=       4 D018508	// W20-3 RH 차종
OR=       4 D018510	// W100 차종 정보
AND LOAD
MPUSH
AND       M1073D	// R07 HD1 (In46) 그리퍼2 파트감지
MOVP      1 D019110	// R07 HD1 G1 Spare4 라인내 잔여수량 카운터
MPOP
AND NOT   M1073D	// R07 HD1 (In46) 그리퍼2 파트감지
MOVP      0 D019110	// R07 HD1 G1 Spare4 라인내 잔여수량 카운터

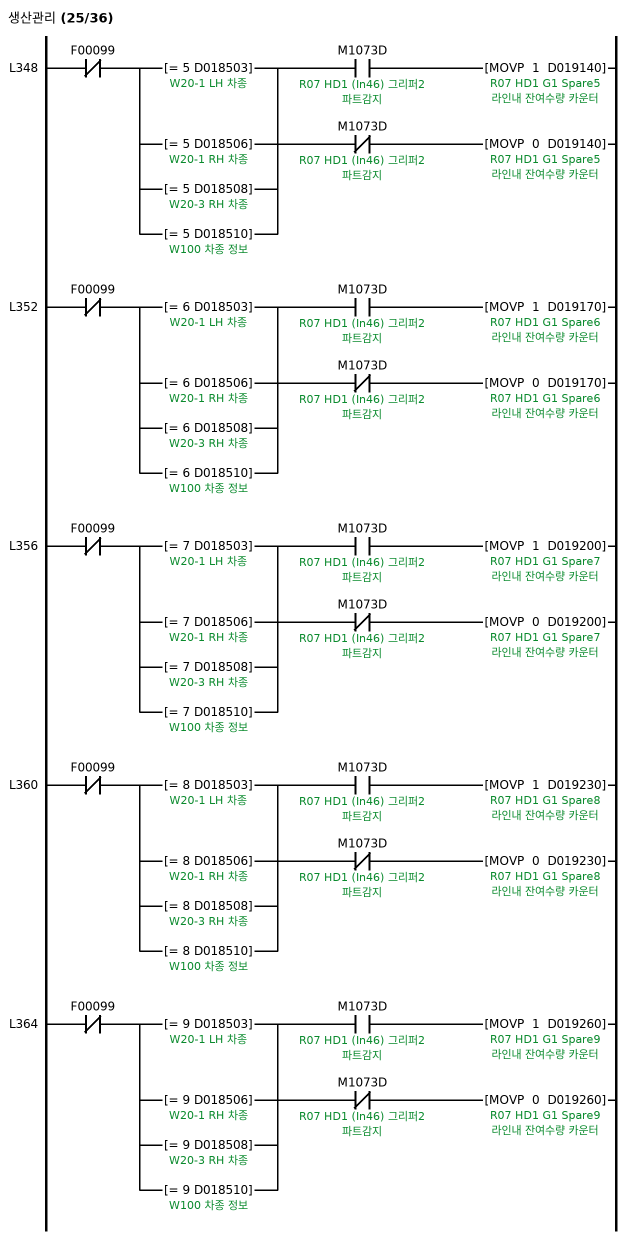
; L348
LOAD NOT  F00099
LOAD=     5 D018503	// W20-1 LH 차종
OR=       5 D018506	// W20-1 RH 차종
OR=       5 D018508	// W20-3 RH 차종
OR=       5 D018510	// W100 차종 정보
AND LOAD
MPUSH
AND       M1073D	// R07 HD1 (In46) 그리퍼2 파트감지
MOVP      1 D019140	// R07 HD1 G1 Spare5 라인내 잔여수량 카운터
MPOP
AND NOT   M1073D	// R07 HD1 (In46) 그리퍼2 파트감지
MOVP      0 D019140	// R07 HD1 G1 Spare5 라인내 잔여수량 카운터
; L352
LOAD NOT  F00099
LOAD=     6 D018503	// W20-1 LH 차종
OR=       6 D018506	// W20-1 RH 차종
OR=       6 D018508	// W20-3 RH 차종
OR=       6 D018510	// W100 차종 정보
AND LOAD
MPUSH
AND       M1073D	// R07 HD1 (In46) 그리퍼2 파트감지
MOVP      1 D019170	// R07 HD1 G1 Spare6 라인내 잔여수량 카운터
MPOP
AND NOT   M1073D	// R07 HD1 (In46) 그리퍼2 파트감지
MOVP      0 D019170	// R07 HD1 G1 Spare6 라인내 잔여수량 카운터
; L356
LOAD NOT  F00099
LOAD=     7 D018503	// W20-1 LH 차종
OR=       7 D018506	// W20-1 RH 차종
OR=       7 D018508	// W20-3 RH 차종
OR=       7 D018510	// W100 차종 정보
AND LOAD
MPUSH
AND       M1073D	// R07 HD1 (In46) 그리퍼2 파트감지
MOVP      1 D019200	// R07 HD1 G1 Spare7 라인내 잔여수량 카운터
MPOP
AND NOT   M1073D	// R07 HD1 (In46) 그리퍼2 파트감지
MOVP      0 D019200	// R07 HD1 G1 Spare7 라인내 잔여수량 카운터
; L360
LOAD NOT  F00099
LOAD=     8 D018503	// W20-1 LH 차종
OR=       8 D018506	// W20-1 RH 차종
OR=       8 D018508	// W20-3 RH 차종
OR=       8 D018510	// W100 차종 정보
AND LOAD
MPUSH
AND       M1073D	// R07 HD1 (In46) 그리퍼2 파트감지
MOVP      1 D019230	// R07 HD1 G1 Spare8 라인내 잔여수량 카운터
MPOP
AND NOT   M1073D	// R07 HD1 (In46) 그리퍼2 파트감지
MOVP      0 D019230	// R07 HD1 G1 Spare8 라인내 잔여수량 카운터
; L364
LOAD NOT  F00099
LOAD=     9 D018503	// W20-1 LH 차종
OR=       9 D018506	// W20-1 RH 차종
OR=       9 D018508	// W20-3 RH 차종
OR=       9 D018510	// W100 차종 정보
AND LOAD
MPUSH
AND       M1073D	// R07 HD1 (In46) 그리퍼2 파트감지
MOVP      1 D019260	// R07 HD1 G1 Spare9 라인내 잔여수량 카운터
MPOP
AND NOT   M1073D	// R07 HD1 (In46) 그리퍼2 파트감지
MOVP      0 D019260	// R07 HD1 G1 Spare9 라인내 잔여수량 카운터

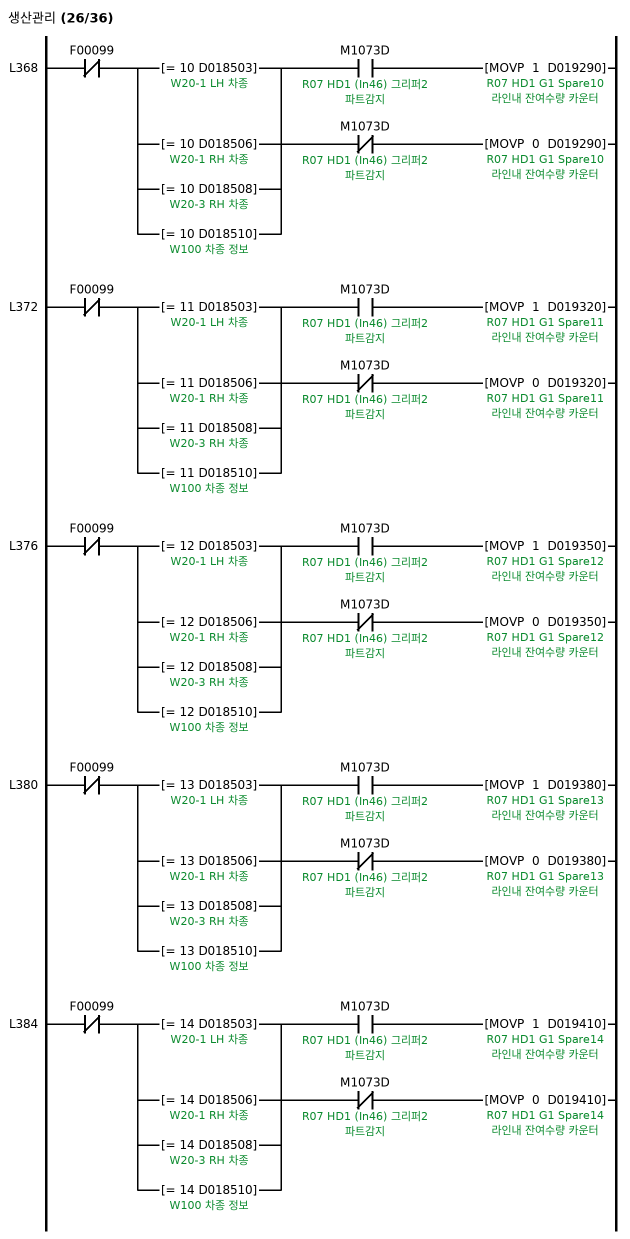
; L368
LOAD NOT  F00099
LOAD=     10 D018503	// W20-1 LH 차종
OR=       10 D018506	// W20-1 RH 차종
OR=       10 D018508	// W20-3 RH 차종
OR=       10 D018510	// W100 차종 정보
AND LOAD
MPUSH
AND       M1073D	// R07 HD1 (In46) 그리퍼2 파트감지
MOVP      1 D019290	// R07 HD1 G1 Spare10 라인내 잔여수량 카운터
MPOP
AND NOT   M1073D	// R07 HD1 (In46) 그리퍼2 파트감지
MOVP      0 D019290	// R07 HD1 G1 Spare10 라인내 잔여수량 카운터
; L372
LOAD NOT  F00099
LOAD=     11 D018503	// W20-1 LH 차종
OR=       11 D018506	// W20-1 RH 차종
OR=       11 D018508	// W20-3 RH 차종
OR=       11 D018510	// W100 차종 정보
AND LOAD
MPUSH
AND       M1073D	// R07 HD1 (In46) 그리퍼2 파트감지
MOVP      1 D019320	// R07 HD1 G1 Spare11 라인내 잔여수량 카운터
MPOP
AND NOT   M1073D	// R07 HD1 (In46) 그리퍼2 파트감지
MOVP      0 D019320	// R07 HD1 G1 Spare11 라인내 잔여수량 카운터
; L376
LOAD NOT  F00099
LOAD=     12 D018503	// W20-1 LH 차종
OR=       12 D018506	// W20-1 RH 차종
OR=       12 D018508	// W20-3 RH 차종
OR=       12 D018510	// W100 차종 정보
AND LOAD
MPUSH
AND       M1073D	// R07 HD1 (In46) 그리퍼2 파트감지
MOVP      1 D019350	// R07 HD1 G1 Spare12 라인내 잔여수량 카운터
MPOP
AND NOT   M1073D	// R07 HD1 (In46) 그리퍼2 파트감지
MOVP      0 D019350	// R07 HD1 G1 Spare12 라인내 잔여수량 카운터
; L380
LOAD NOT  F00099
LOAD=     13 D018503	// W20-1 LH 차종
OR=       13 D018506	// W20-1 RH 차종
OR=       13 D018508	// W20-3 RH 차종
OR=       13 D018510	// W100 차종 정보
AND LOAD
MPUSH
AND       M1073D	// R07 HD1 (In46) 그리퍼2 파트감지
MOVP      1 D019380	// R07 HD1 G1 Spare13 라인내 잔여수량 카운터
MPOP
AND NOT   M1073D	// R07 HD1 (In46) 그리퍼2 파트감지
MOVP      0 D019380	// R07 HD1 G1 Spare13 라인내 잔여수량 카운터
; L384
LOAD NOT  F00099
LOAD=     14 D018503	// W20-1 LH 차종
OR=       14 D018506	// W20-1 RH 차종
OR=       14 D018508	// W20-3 RH 차종
OR=       14 D018510	// W100 차종 정보
AND LOAD
MPUSH
AND       M1073D	// R07 HD1 (In46) 그리퍼2 파트감지
MOVP      1 D019410	// R07 HD1 G1 Spare14 라인내 잔여수량 카운터
MPOP
AND NOT   M1073D	// R07 HD1 (In46) 그리퍼2 파트감지
MOVP      0 D019410	// R07 HD1 G1 Spare14 라인내 잔여수량 카운터

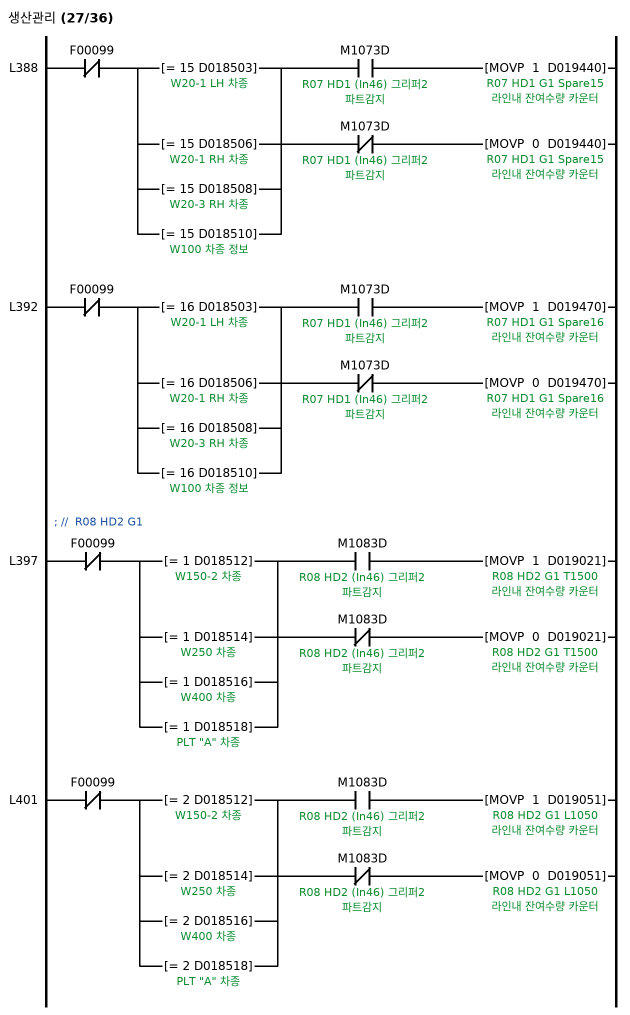
; L388
LOAD NOT  F00099
LOAD=     15 D018503	// W20-1 LH 차종
OR=       15 D018506	// W20-1 RH 차종
OR=       15 D018508	// W20-3 RH 차종
OR=       15 D018510	// W100 차종 정보
AND LOAD
MPUSH
AND       M1073D	// R07 HD1 (In46) 그리퍼2 파트감지
MOVP      1 D019440	// R07 HD1 G1 Spare15 라인내 잔여수량 카운터
MPOP
AND NOT   M1073D	// R07 HD1 (In46) 그리퍼2 파트감지
MOVP      0 D019440	// R07 HD1 G1 Spare15 라인내 잔여수량 카운터
; L392
LOAD NOT  F00099
LOAD=     16 D018503	// W20-1 LH 차종
OR=       16 D018506	// W20-1 RH 차종
OR=       16 D018508	// W20-3 RH 차종
OR=       16 D018510	// W100 차종 정보
AND LOAD
MPUSH
AND       M1073D	// R07 HD1 (In46) 그리퍼2 파트감지
MOVP      1 D019470	// R07 HD1 G1 Spare16 라인내 잔여수량 카운터
MPOP
AND NOT   M1073D	// R07 HD1 (In46) 그리퍼2 파트감지
MOVP      0 D019470	// R07 HD1 G1 Spare16 라인내 잔여수량 카운터
//   //  R08 HD2 G1
; L397
LOAD NOT  F00099
LOAD=     1 D018512	// W150-2 차종
OR=       1 D018514	// W250 차종
OR=       1 D018516	// W400 차종
OR=       1 D018518	// PLT "A" 차종
AND LOAD
MPUSH
AND       M1083D	// R08 HD2 (In46) 그리퍼2 파트감지
MOVP      1 D019021	// R08 HD2 G1 T1500 라인내 잔여수량 카운터
MPOP
AND NOT   M1083D	// R08 HD2 (In46) 그리퍼2 파트감지
MOVP      0 D019021	// R08 HD2 G1 T1500 라인내 잔여수량 카운터
; L401
LOAD NOT  F00099
LOAD=     2 D018512	// W150-2 차종
OR=       2 D018514	// W250 차종
OR=       2 D018516	// W400 차종
OR=       2 D018518	// PLT "A" 차종
AND LOAD
MPUSH
AND       M1083D	// R08 HD2 (In46) 그리퍼2 파트감지
MOVP      1 D019051	// R08 HD2 G1 L1050 라인내 잔여수량 카운터
MPOP
AND NOT   M1083D	// R08 HD2 (In46) 그리퍼2 파트감지
MOVP      0 D019051	// R08 HD2 G1 L1050 라인내 잔여수량 카운터

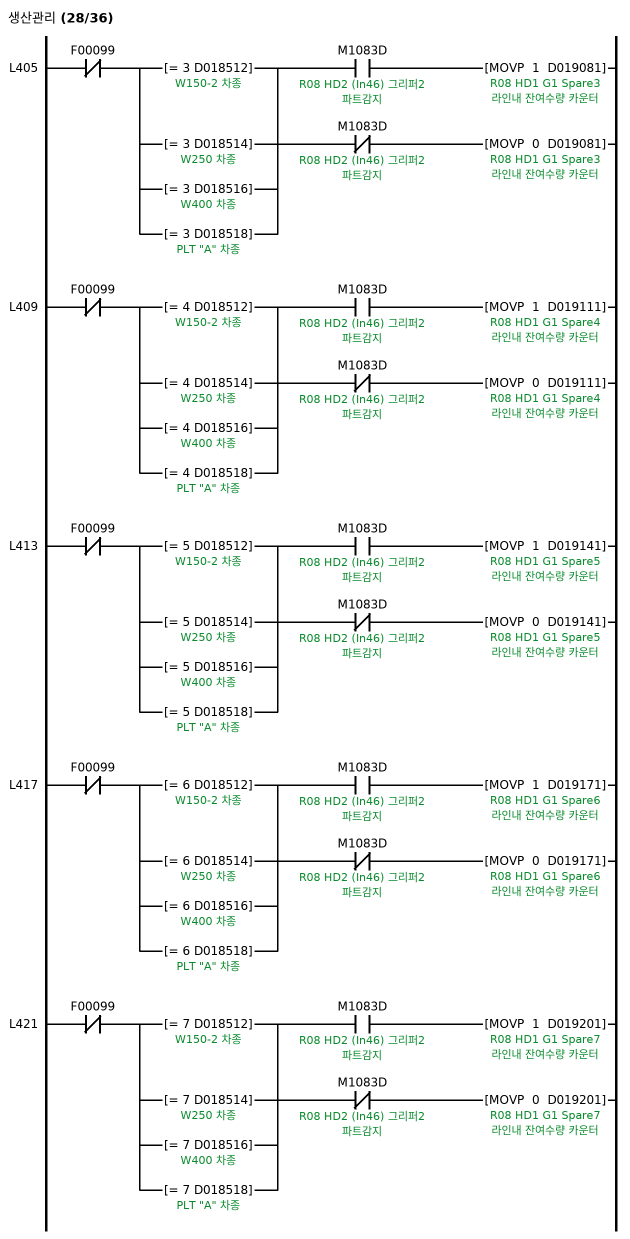
; L405
LOAD NOT  F00099
LOAD=     3 D018512	// W150-2 차종
OR=       3 D018514	// W250 차종
OR=       3 D018516	// W400 차종
OR=       3 D018518	// PLT "A" 차종
AND LOAD
MPUSH
AND       M1083D	// R08 HD2 (In46) 그리퍼2 파트감지
MOVP      1 D019081	// R08 HD1 G1 Spare3 라인내 잔여수량 카운터
MPOP
AND NOT   M1083D	// R08 HD2 (In46) 그리퍼2 파트감지
MOVP      0 D019081	// R08 HD1 G1 Spare3 라인내 잔여수량 카운터
; L409
LOAD NOT  F00099
LOAD=     4 D018512	// W150-2 차종
OR=       4 D018514	// W250 차종
OR=       4 D018516	// W400 차종
OR=       4 D018518	// PLT "A" 차종
AND LOAD
MPUSH
AND       M1083D	// R08 HD2 (In46) 그리퍼2 파트감지
MOVP      1 D019111	// R08 HD1 G1 Spare4 라인내 잔여수량 카운터
MPOP
AND NOT   M1083D	// R08 HD2 (In46) 그리퍼2 파트감지
MOVP      0 D019111	// R08 HD1 G1 Spare4 라인내 잔여수량 카운터
; L413
LOAD NOT  F00099
LOAD=     5 D018512	// W150-2 차종
OR=       5 D018514	// W250 차종
OR=       5 D018516	// W400 차종
OR=       5 D018518	// PLT "A" 차종
AND LOAD
MPUSH
AND       M1083D	// R08 HD2 (In46) 그리퍼2 파트감지
MOVP      1 D019141	// R08 HD1 G1 Spare5 라인내 잔여수량 카운터
MPOP
AND NOT   M1083D	// R08 HD2 (In46) 그리퍼2 파트감지
MOVP      0 D019141	// R08 HD1 G1 Spare5 라인내 잔여수량 카운터
; L417
LOAD NOT  F00099
LOAD=     6 D018512	// W150-2 차종
OR=       6 D018514	// W250 차종
OR=       6 D018516	// W400 차종
OR=       6 D018518	// PLT "A" 차종
AND LOAD
MPUSH
AND       M1083D	// R08 HD2 (In46) 그리퍼2 파트감지
MOVP      1 D019171	// R08 HD1 G1 Spare6 라인내 잔여수량 카운터
MPOP
AND NOT   M1083D	// R08 HD2 (In46) 그리퍼2 파트감지
MOVP      0 D019171	// R08 HD1 G1 Spare6 라인내 잔여수량 카운터
; L421
LOAD NOT  F00099
LOAD=     7 D018512	// W150-2 차종
OR=       7 D018514	// W250 차종
OR=       7 D018516	// W400 차종
OR=       7 D018518	// PLT "A" 차종
AND LOAD
MPUSH
AND       M1083D	// R08 HD2 (In46) 그리퍼2 파트감지
MOVP      1 D019201	// R08 HD1 G1 Spare7 라인내 잔여수량 카운터
MPOP
AND NOT   M1083D	// R08 HD2 (In46) 그리퍼2 파트감지
MOVP      0 D019201	// R08 HD1 G1 Spare7 라인내 잔여수량 카운터

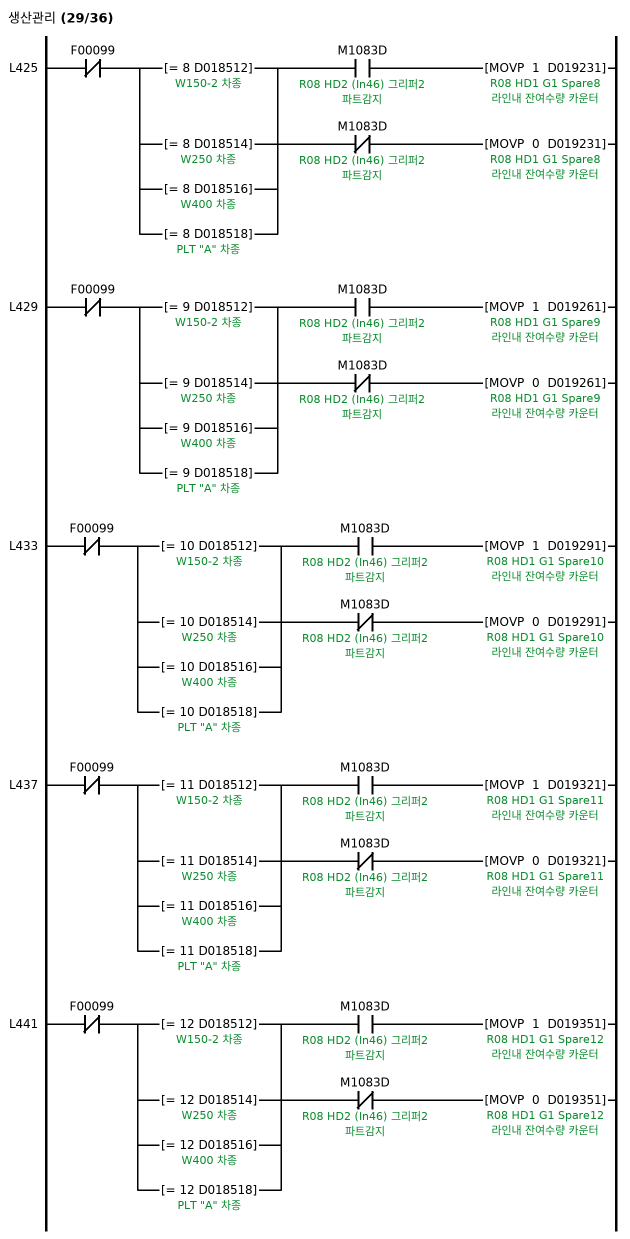
; L425
LOAD NOT  F00099
LOAD=     8 D018512	// W150-2 차종
OR=       8 D018514	// W250 차종
OR=       8 D018516	// W400 차종
OR=       8 D018518	// PLT "A" 차종
AND LOAD
MPUSH
AND       M1083D	// R08 HD2 (In46) 그리퍼2 파트감지
MOVP      1 D019231	// R08 HD1 G1 Spare8 라인내 잔여수량 카운터
MPOP
AND NOT   M1083D	// R08 HD2 (In46) 그리퍼2 파트감지
MOVP      0 D019231	// R08 HD1 G1 Spare8 라인내 잔여수량 카운터
; L429
LOAD NOT  F00099
LOAD=     9 D018512	// W150-2 차종
OR=       9 D018514	// W250 차종
OR=       9 D018516	// W400 차종
OR=       9 D018518	// PLT "A" 차종
AND LOAD
MPUSH
AND       M1083D	// R08 HD2 (In46) 그리퍼2 파트감지
MOVP      1 D019261	// R08 HD1 G1 Spare9 라인내 잔여수량 카운터
MPOP
AND NOT   M1083D	// R08 HD2 (In46) 그리퍼2 파트감지
MOVP      0 D019261	// R08 HD1 G1 Spare9 라인내 잔여수량 카운터
; L433
LOAD NOT  F00099
LOAD=     10 D018512	// W150-2 차종
OR=       10 D018514	// W250 차종
OR=       10 D018516	// W400 차종
OR=       10 D018518	// PLT "A" 차종
AND LOAD
MPUSH
AND       M1083D	// R08 HD2 (In46) 그리퍼2 파트감지
MOVP      1 D019291	// R08 HD1 G1 Spare10 라인내 잔여수량 카운터
MPOP
AND NOT   M1083D	// R08 HD2 (In46) 그리퍼2 파트감지
MOVP      0 D019291	// R08 HD1 G1 Spare10 라인내 잔여수량 카운터
; L437
LOAD NOT  F00099
LOAD=     11 D018512	// W150-2 차종
OR=       11 D018514	// W250 차종
OR=       11 D018516	// W400 차종
OR=       11 D018518	// PLT "A" 차종
AND LOAD
MPUSH
AND       M1083D	// R08 HD2 (In46) 그리퍼2 파트감지
MOVP      1 D019321	// R08 HD1 G1 Spare11 라인내 잔여수량 카운터
MPOP
AND NOT   M1083D	// R08 HD2 (In46) 그리퍼2 파트감지
MOVP      0 D019321	// R08 HD1 G1 Spare11 라인내 잔여수량 카운터
; L441
LOAD NOT  F00099
LOAD=     12 D018512	// W150-2 차종
OR=       12 D018514	// W250 차종
OR=       12 D018516	// W400 차종
OR=       12 D018518	// PLT "A" 차종
AND LOAD
MPUSH
AND       M1083D	// R08 HD2 (In46) 그리퍼2 파트감지
MOVP      1 D019351	// R08 HD1 G1 Spare12 라인내 잔여수량 카운터
MPOP
AND NOT   M1083D	// R08 HD2 (In46) 그리퍼2 파트감지
MOVP      0 D019351	// R08 HD1 G1 Spare12 라인내 잔여수량 카운터

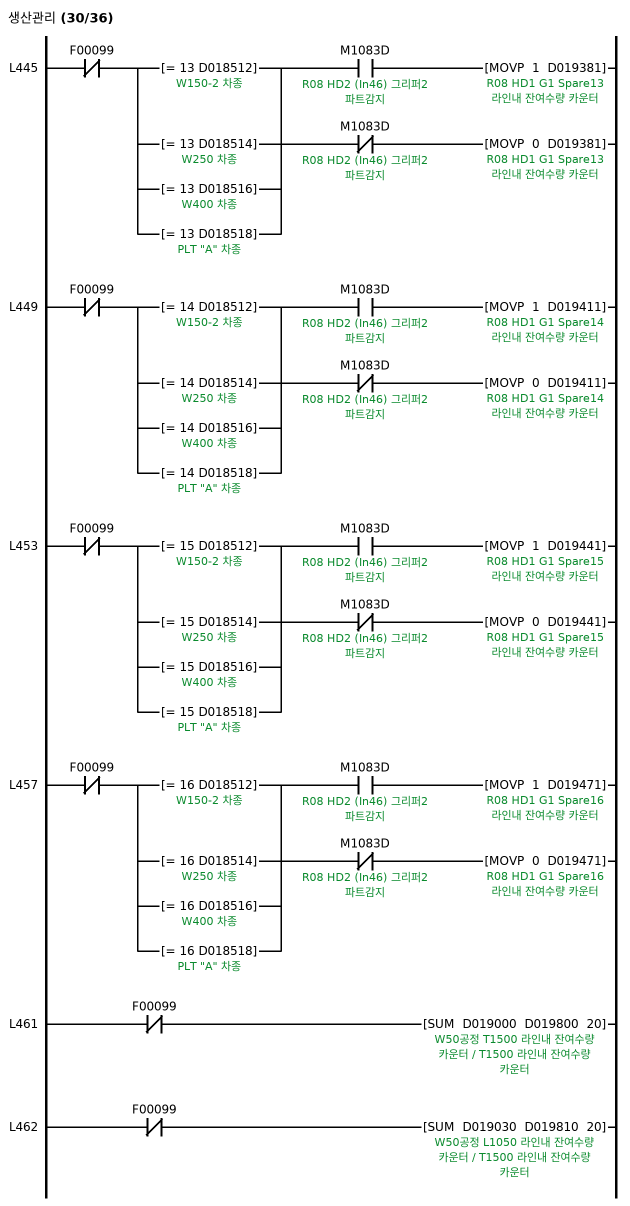
; L445
LOAD NOT  F00099
LOAD=     13 D018512	// W150-2 차종
OR=       13 D018514	// W250 차종
OR=       13 D018516	// W400 차종
OR=       13 D018518	// PLT "A" 차종
AND LOAD
MPUSH
AND       M1083D	// R08 HD2 (In46) 그리퍼2 파트감지
MOVP      1 D019381	// R08 HD1 G1 Spare13 라인내 잔여수량 카운터
MPOP
AND NOT   M1083D	// R08 HD2 (In46) 그리퍼2 파트감지
MOVP      0 D019381	// R08 HD1 G1 Spare13 라인내 잔여수량 카운터
; L449
LOAD NOT  F00099
LOAD=     14 D018512	// W150-2 차종
OR=       14 D018514	// W250 차종
OR=       14 D018516	// W400 차종
OR=       14 D018518	// PLT "A" 차종
AND LOAD
MPUSH
AND       M1083D	// R08 HD2 (In46) 그리퍼2 파트감지
MOVP      1 D019411	// R08 HD1 G1 Spare14 라인내 잔여수량 카운터
MPOP
AND NOT   M1083D	// R08 HD2 (In46) 그리퍼2 파트감지
MOVP      0 D019411	// R08 HD1 G1 Spare14 라인내 잔여수량 카운터
; L453
LOAD NOT  F00099
LOAD=     15 D018512	// W150-2 차종
OR=       15 D018514	// W250 차종
OR=       15 D018516	// W400 차종
OR=       15 D018518	// PLT "A" 차종
AND LOAD
MPUSH
AND       M1083D	// R08 HD2 (In46) 그리퍼2 파트감지
MOVP      1 D019441	// R08 HD1 G1 Spare15 라인내 잔여수량 카운터
MPOP
AND NOT   M1083D	// R08 HD2 (In46) 그리퍼2 파트감지
MOVP      0 D019441	// R08 HD1 G1 Spare15 라인내 잔여수량 카운터
; L457
LOAD NOT  F00099
LOAD=     16 D018512	// W150-2 차종
OR=       16 D018514	// W250 차종
OR=       16 D018516	// W400 차종
OR=       16 D018518	// PLT "A" 차종
AND LOAD
MPUSH
AND       M1083D	// R08 HD2 (In46) 그리퍼2 파트감지
MOVP      1 D019471	// R08 HD1 G1 Spare16 라인내 잔여수량 카운터
MPOP
AND NOT   M1083D	// R08 HD2 (In46) 그리퍼2 파트감지
MOVP      0 D019471	// R08 HD1 G1 Spare16 라인내 잔여수량 카운터
; L461
LOAD NOT  F00099
SUM       D019000 D019800 20	// W50공정 T1500 라인내 잔여수량 카운터 / T1500 라인내 잔여수량 카운터
; L462
LOAD NOT  F00099
SUM       D019030 D019810 20	// W50공정 L1050 라인내 잔여수량 카운터 / T1500 라인내 잔여수량 카운터

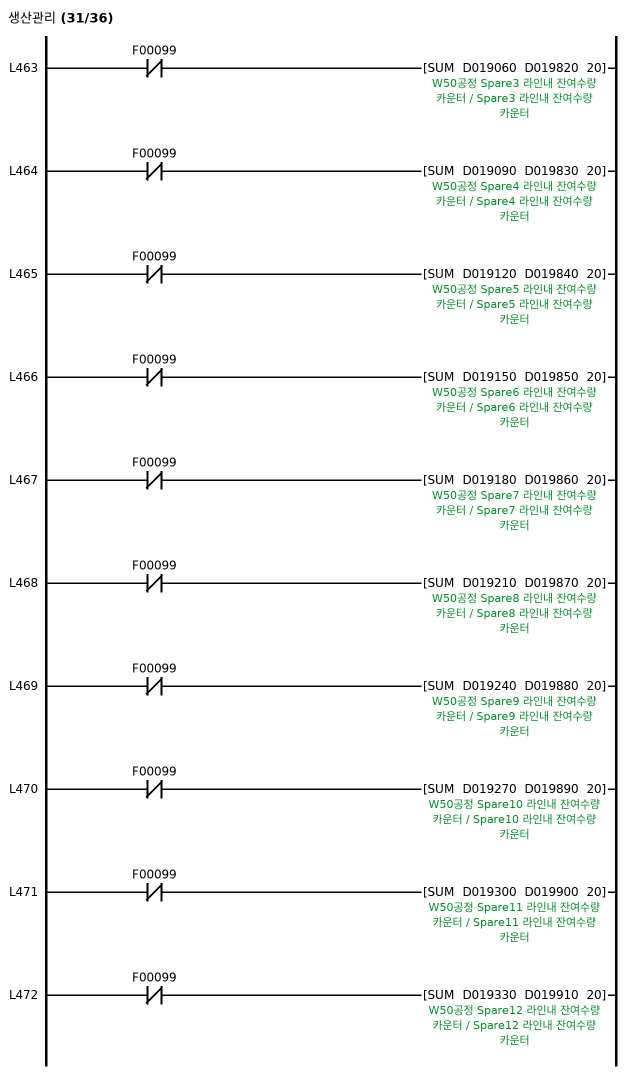
; L463
LOAD NOT  F00099
SUM       D019060 D019820 20	// W50공정 Spare3 라인내 잔여수량 카운터 / Spare3 라인내 잔여수량 카운터
; L464
LOAD NOT  F00099
SUM       D019090 D019830 20	// W50공정 Spare4 라인내 잔여수량 카운터 / Spare4 라인내 잔여수량 카운터
; L465
LOAD NOT  F00099
SUM       D019120 D019840 20	// W50공정 Spare5 라인내 잔여수량 카운터 / Spare5 라인내 잔여수량 카운터
; L466
LOAD NOT  F00099
SUM       D019150 D019850 20	// W50공정 Spare6 라인내 잔여수량 카운터 / Spare6 라인내 잔여수량 카운터
; L467
LOAD NOT  F00099
SUM       D019180 D019860 20	// W50공정 Spare7 라인내 잔여수량 카운터 / Spare7 라인내 잔여수량 카운터
; L468
LOAD NOT  F00099
SUM       D019210 D019870 20	// W50공정 Spare8 라인내 잔여수량 카운터 / Spare8 라인내 잔여수량 카운터
; L469
LOAD NOT  F00099
SUM       D019240 D019880 20	// W50공정 Spare9 라인내 잔여수량 카운터 / Spare9 라인내 잔여수량 카운터
; L470
LOAD NOT  F00099
SUM       D019270 D019890 20	// W50공정 Spare10 라인내 잔여수량 카운터 / Spare10 라인내 잔여수량 카운터
; L471
LOAD NOT  F00099
SUM       D019300 D019900 20	// W50공정 Spare11 라인내 잔여수량 카운터 / Spare11 라인내 잔여수량 카운터
; L472
LOAD NOT  F00099
SUM       D019330 D019910 20	// W50공정 Spare12 라인내 잔여수량 카운터 / Spare12 라인내 잔여수량 카운터

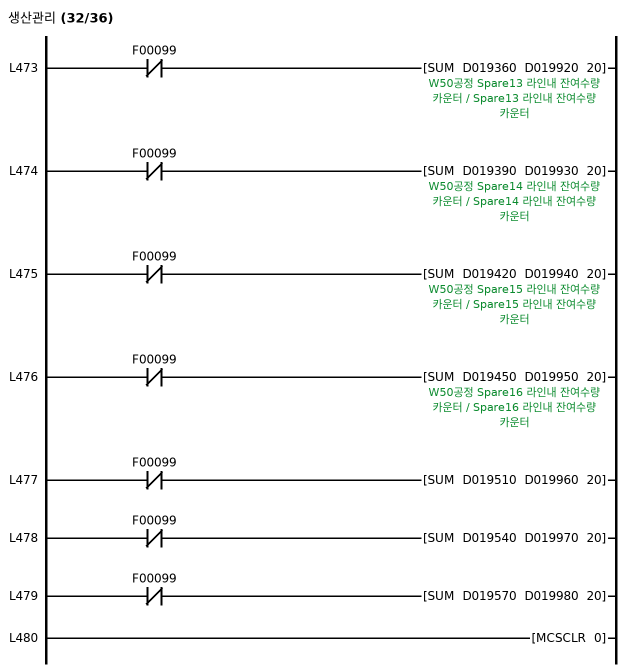
; L473
LOAD NOT  F00099
SUM       D019360 D019920 20	// W50공정 Spare13 라인내 잔여수량 카운터 / Spare13 라인내 잔여수량 카운터
; L474
LOAD NOT  F00099
SUM       D019390 D019930 20	// W50공정 Spare14 라인내 잔여수량 카운터 / Spare14 라인내 잔여수량 카운터
; L475
LOAD NOT  F00099
SUM       D019420 D019940 20	// W50공정 Spare15 라인내 잔여수량 카운터 / Spare15 라인내 잔여수량 카운터
; L476
LOAD NOT  F00099
SUM       D019450 D019950 20	// W50공정 Spare16 라인내 잔여수량 카운터 / Spare16 라인내 잔여수량 카운터
; L477
LOAD NOT  F00099
SUM       D019510 D019960 20
; L478
LOAD NOT  F00099
SUM       D019540 D019970 20
; L479
LOAD NOT  F00099
SUM       D019570 D019980 20
; L480
MCSCLR    0

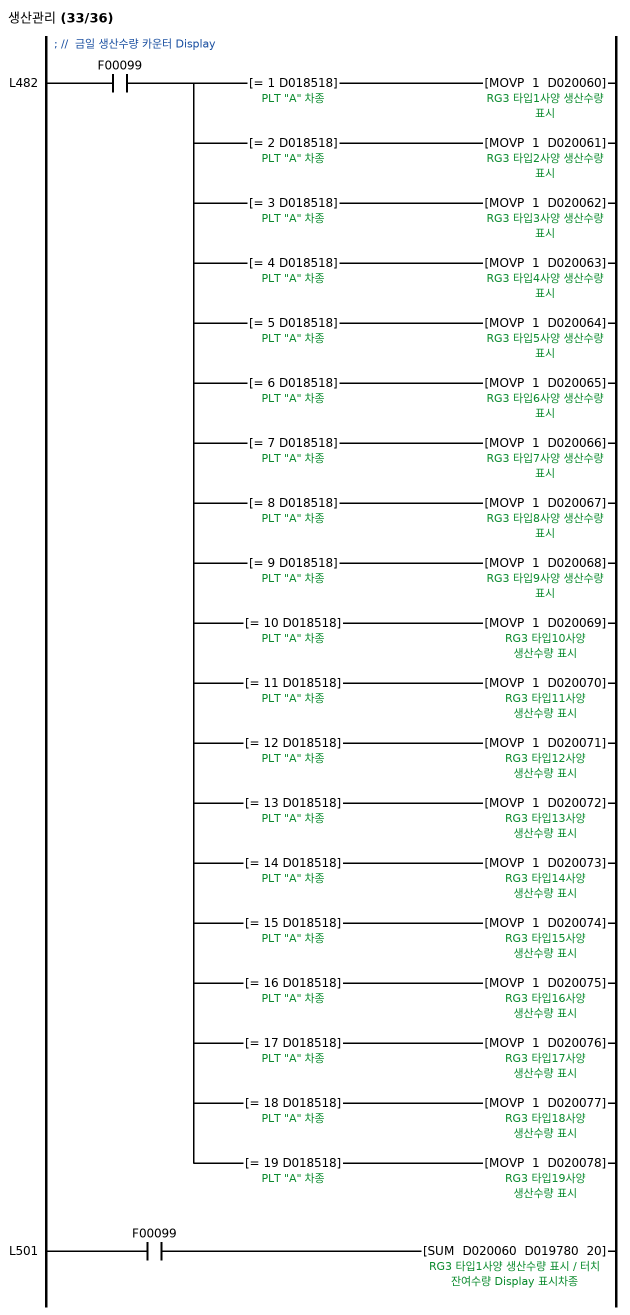
//   //  금일 생산수량 카운터 Display
; L482
LOAD      F00099
MPUSH
AND=      1 D018518	// PLT "A" 차종
MOVP      1 D020060	// RG3 타입1사양 생산수량 표시
MLOAD
AND=      2 D018518	// PLT "A" 차종
MOVP      1 D020061	// RG3 타입2사양 생산수량 표시
MLOAD
AND=      3 D018518	// PLT "A" 차종
MOVP      1 D020062	// RG3 타입3사양 생산수량 표시
MLOAD
AND=      4 D018518	// PLT "A" 차종
MOVP      1 D020063	// RG3 타입4사양 생산수량 표시
MLOAD
AND=      5 D018518	// PLT "A" 차종
MOVP      1 D020064	// RG3 타입5사양 생산수량 표시
MLOAD
AND=      6 D018518	// PLT "A" 차종
MOVP      1 D020065	// RG3 타입6사양 생산수량 표시
MLOAD
AND=      7 D018518	// PLT "A" 차종
MOVP      1 D020066	// RG3 타입7사양 생산수량 표시
MLOAD
AND=      8 D018518	// PLT "A" 차종
MOVP      1 D020067	// RG3 타입8사양 생산수량 표시
MLOAD
AND=      9 D018518	// PLT "A" 차종
MOVP      1 D020068	// RG3 타입9사양 생산수량 표시
MLOAD
AND=      10 D018518	// PLT "A" 차종
MOVP      1 D020069	// RG3 타입10사양 생산수량 표시
MLOAD
AND=      11 D018518	// PLT "A" 차종
MOVP      1 D020070	// RG3 타입11사양 생산수량 표시
MLOAD
AND=      12 D018518	// PLT "A" 차종
MOVP      1 D020071	// RG3 타입12사양 생산수량 표시
MLOAD
AND=      13 D018518	// PLT "A" 차종
MOVP      1 D020072	// RG3 타입13사양 생산수량 표시
MLOAD
AND=      14 D018518	// PLT "A" 차종
MOVP      1 D020073	// RG3 타입14사양 생산수량 표시
MLOAD
AND=      15 D018518	// PLT "A" 차종
MOVP      1 D020074	// RG3 타입15사양 생산수량 표시
MLOAD
AND=      16 D018518	// PLT "A" 차종
MOVP      1 D020075	// RG3 타입16사양 생산수량 표시
MLOAD
AND=      17 D018518	// PLT "A" 차종
MOVP      1 D020076	// RG3 타입17사양 생산수량 표시
MLOAD
AND=      18 D018518	// PLT "A" 차종
MOVP      1 D020077	// RG3 타입18사양 생산수량 표시
MPOP
AND=      19 D018518	// PLT "A" 차종
MOVP      1 D020078	// RG3 타입19사양 생산수량 표시
; L501
LOAD      F00099
SUM       D020060 D019780 20	// RG3 타입1사양 생산수량 표시 / 터치 잔여수량 Display 표시차종

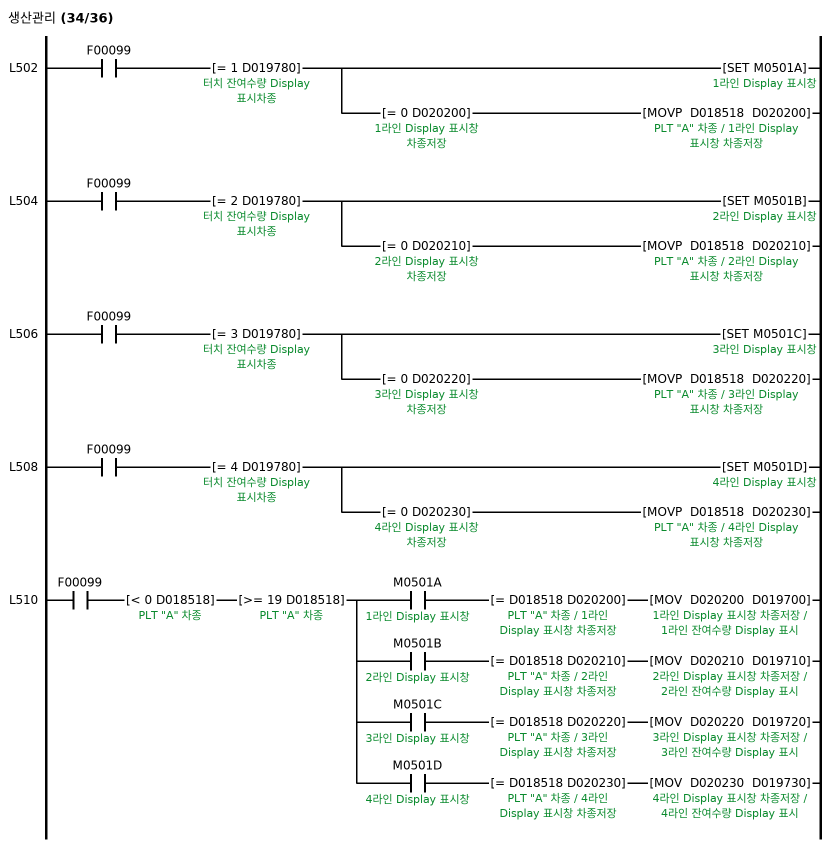
; L502
LOAD      F00099
AND=      1 D019780	// 터치 잔여수량 Display 표시차종
SET       M0501A	// 1라인 Display 표시창
AND=      0 D020200	// 1라인 Display 표시창 차종저장
MOVP      D018518 D020200	// PLT "A" 차종 / 1라인 Display 표시창 차종저장
; L504
LOAD      F00099
AND=      2 D019780	// 터치 잔여수량 Display 표시차종
SET       M0501B	// 2라인 Display 표시창
AND=      0 D020210	// 2라인 Display 표시창 차종저장
MOVP      D018518 D020210	// PLT "A" 차종 / 2라인 Display 표시창 차종저장
; L506
LOAD      F00099
AND=      3 D019780	// 터치 잔여수량 Display 표시차종
SET       M0501C	// 3라인 Display 표시창
AND=      0 D020220	// 3라인 Display 표시창 차종저장
MOVP      D018518 D020220	// PLT "A" 차종 / 3라인 Display 표시창 차종저장
; L508
LOAD      F00099
AND=      4 D019780	// 터치 잔여수량 Display 표시차종
SET       M0501D	// 4라인 Display 표시창
AND=      0 D020230	// 4라인 Display 표시창 차종저장
MOVP      D018518 D020230	// PLT "A" 차종 / 4라인 Display 표시창 차종저장
; L510
LOAD      F00099
AND<      0 D018518	// PLT "A" 차종
AND>=     19 D018518	// PLT "A" 차종
MPUSH
AND       M0501A	// 1라인 Display 표시창
AND=      D018518 D020200	// PLT "A" 차종 / 1라인 Display 표시창 차종저장
MOV       D020200 D019700	// 1라인 Display 표시창 차종저장 / 1라인 잔여수량 Display 표시 
MLOAD
AND       M0501B	// 2라인 Display 표시창
AND=      D018518 D020210	// PLT "A" 차종 / 2라인 Display 표시창 차종저장
MOV       D020210 D019710	// 2라인 Display 표시창 차종저장 / 2라인 잔여수량 Display 표시 
MLOAD
AND       M0501C	// 3라인 Display 표시창
AND=      D018518 D020220	// PLT "A" 차종 / 3라인 Display 표시창 차종저장
MOV       D020220 D019720	// 3라인 Display 표시창 차종저장 / 3라인 잔여수량 Display 표시 
MPOP
AND       M0501D	// 4라인 Display 표시창
AND=      D018518 D020230	// PLT "A" 차종 / 4라인 Display 표시창 차종저장
MOV       D020230 D019730	// 4라인 Display 표시창 차종저장 / 4라인 잔여수량 Display 표시 

